Yaskawa INFORM job: A_ROOF_UPPER_0614_2_PAINT_10.JBI

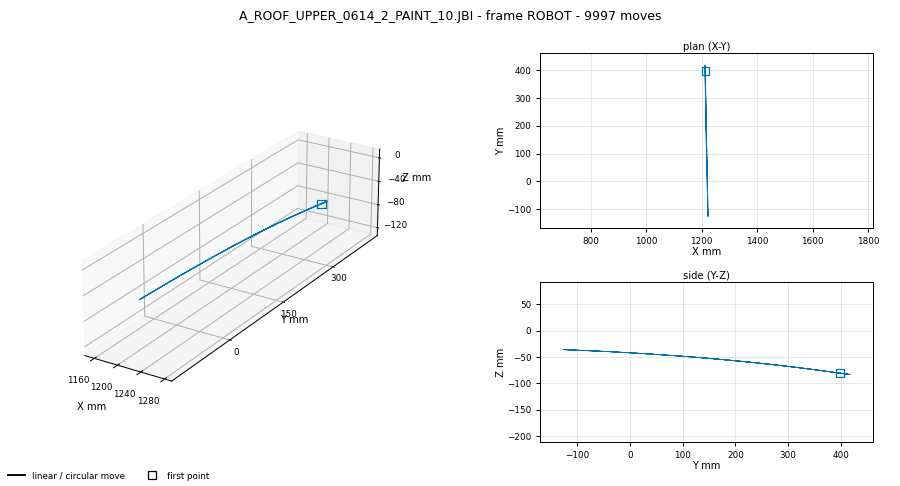
[picture p0: tool path of A_ROOF_UPPER_0614_2_PAINT_10.JBI in frame ROBOT, 9997 of 9997 moves have a stored position in this frame; points joined in program order, loops and branches not executed]
/JOB
//NAME A_ROOF_UPPER_0614_2_PAINT10
//POS
///NPOS 9997,0,0,0,0,0
///TOOL 1
///USER 0
///POSTYPE ROBOT
///RECTAN
///RCONF 1,0,0,0,0,0,0,0,0,0,0,0,0,0,0,0,0,0,0,0,0,0,0,0
C00000=1214.064,397.610,-80.249,-175.800,8.118,148.366
C00001=1214.059,397.858,-80.283,-175.800,8.120,148.367
C00002=1214.055,398.106,-80.318,-175.799,8.123,148.367
C00003=1214.051,398.353,-80.352,-175.799,8.125,148.368
C00004=1214.047,398.601,-80.386,-175.799,8.128,148.368
C00005=1214.043,398.849,-80.421,-175.797,8.130,148.369
C00006=1214.038,399.096,-80.456,-175.797,8.133,148.369
C00007=1214.035,399.343,-80.491,-175.796,8.135,148.370
C00008=1214.031,399.591,-80.525,-175.796,8.138,148.370
C00009=1214.027,399.839,-80.560,-175.795,8.140,148.371
C00010=1214.022,400.086,-80.594,-175.794,8.143,148.371
C00011=1214.019,400.334,-80.629,-175.794,8.145,148.372
C00012=1214.014,400.581,-80.663,-175.794,8.147,148.372
C00013=1214.010,400.830,-80.698,-175.793,8.150,148.373
C00014=1214.007,401.076,-80.732,-175.792,8.152,148.373
C00015=1214.003,401.324,-80.767,-175.792,8.154,148.373
C00016=1213.998,401.572,-80.802,-175.791,8.157,148.374
C00017=1213.994,401.819,-80.836,-175.791,8.159,148.374
C00018=1213.991,402.067,-80.870,-175.790,8.162,148.375
C00019=1213.986,402.314,-80.905,-175.790,8.164,148.375
C00020=1213.982,402.562,-80.940,-175.789,8.167,148.376
C00021=1213.978,402.809,-80.975,-175.788,8.169,148.376
C00022=1213.975,403.057,-81.009,-175.788,8.171,148.377
C00023=1213.970,403.304,-81.044,-175.787,8.174,148.377
C00024=1213.966,403.552,-81.079,-175.787,8.176,148.378
C00025=1213.962,403.799,-81.114,-175.787,8.178,148.378
C00026=1213.958,404.047,-81.149,-175.786,8.180,148.379
C00027=1213.954,404.295,-81.182,-175.785,8.183,148.379
C00028=1213.950,404.543,-81.217,-175.784,8.185,148.380
C00029=1213.946,404.789,-81.252,-175.784,8.188,148.380
C00030=1213.942,405.038,-81.287,-175.784,8.190,148.381
C00031=1213.937,405.285,-81.322,-175.783,8.192,148.381
C00032=1213.934,405.532,-81.357,-175.783,8.195,148.382
C00033=1213.930,405.780,-81.391,-175.782,8.197,148.382
C00034=1213.926,406.028,-81.426,-175.782,8.199,148.382
C00035=1213.921,406.275,-81.460,-175.782,8.202,148.383
C00036=1213.918,406.523,-81.496,-175.781,8.204,148.383
C00037=1213.914,406.770,-81.530,-175.780,8.207,148.384
C00038=1213.910,407.018,-81.565,-175.780,8.209,148.384
C00039=1213.905,407.265,-81.600,-175.779,8.211,148.385
C00040=1213.901,407.513,-81.635,-175.779,8.213,148.385
C00041=1213.897,407.760,-81.669,-175.778,8.215,148.386
C00042=1213.894,408.007,-81.704,-175.778,8.217,148.386
C00043=1213.890,408.256,-81.739,-175.777,8.220,148.387
C00044=1213.885,408.503,-81.773,-175.777,8.223,148.387
C00045=1213.882,408.750,-81.809,-175.776,8.224,148.387
C00046=1213.877,408.998,-81.843,-175.776,8.227,148.388
C00047=1213.873,409.246,-81.878,-175.776,8.229,148.388
C00048=1213.869,409.493,-81.913,-175.775,8.231,148.389
C00049=1213.866,409.741,-81.948,-175.775,8.233,148.389
C00050=1213.861,409.988,-81.982,-175.774,8.236,148.390
C00051=1213.858,410.236,-82.018,-175.774,8.238,148.390
C00052=1213.853,410.483,-82.052,-175.773,8.240,148.391
C00053=1213.849,410.730,-82.088,-175.773,8.243,148.391
C00054=1213.845,410.979,-82.123,-175.772,8.245,148.392
C00055=1213.841,411.226,-82.157,-175.772,8.247,148.392
C00056=1213.837,411.474,-82.193,-175.772,8.249,148.393
C00057=1213.833,411.721,-82.226,-175.771,8.251,148.393
C00058=1213.830,411.968,-82.262,-175.771,8.253,148.393
C00059=1213.825,412.216,-82.296,-175.770,8.255,148.394
C00060=1213.821,412.464,-82.331,-175.770,8.258,148.394
C00061=1213.817,412.710,-82.366,-175.770,8.260,148.395
C00062=1213.813,412.959,-82.401,-175.768,8.263,148.395
C00063=1213.809,413.206,-82.437,-175.768,8.265,148.396
C00064=1213.805,413.454,-82.471,-175.768,8.267,148.396
C00065=1213.801,413.701,-82.507,-175.767,8.269,148.397
C00066=1213.796,413.948,-82.541,-175.767,8.271,148.397
C00067=1213.793,414.196,-82.577,-175.767,8.273,148.398
C00068=1213.789,414.443,-82.611,-175.766,8.275,148.398
C00069=1213.785,414.691,-82.646,-175.766,8.278,148.398
C00070=1213.781,414.939,-82.681,-175.765,8.280,148.399
C00071=1213.777,415.186,-82.716,-175.765,8.282,148.399
C00072=1213.773,415.424,-82.750,-175.764,8.284,148.400
C00073=1213.769,415.662,-82.783,-175.764,8.286,148.400
C00074=1213.766,415.900,-82.817,-175.763,8.288,148.400
C00075=1213.761,416.139,-82.851,-175.763,8.290,148.401
C00076=1213.757,416.377,-82.885,-175.763,8.292,148.401
C00077=1213.754,416.616,-82.918,-175.763,8.294,148.402
C00078=1213.752,416.853,-82.951,-175.762,8.296,148.402
C00079=1213.753,417.091,-82.985,-175.762,8.298,148.403
C00080=1213.331,417.091,-83.021,-175.765,8.308,148.406
C00081=1213.330,416.852,-82.988,-175.765,8.306,148.406
C00082=1213.332,416.612,-82.954,-175.766,8.304,148.406
C00083=1213.336,416.372,-82.920,-175.766,8.302,148.405
C00084=1213.339,416.134,-82.886,-175.766,8.301,148.405
C00085=1213.343,415.894,-82.852,-175.767,8.299,148.404
C00086=1213.348,415.655,-82.818,-175.767,8.297,148.404
C00087=1213.351,415.415,-82.785,-175.768,8.295,148.403
C00088=1213.355,415.175,-82.750,-175.768,8.293,148.403
C00089=1213.359,414.928,-82.715,-175.768,8.290,148.402
C00090=1213.363,414.680,-82.680,-175.769,8.288,148.402
C00091=1213.367,414.433,-82.645,-175.769,8.286,148.402
C00092=1213.371,414.185,-82.610,-175.769,8.284,148.401
C00093=1213.376,413.938,-82.576,-175.770,8.282,148.401
C00094=1213.379,413.690,-82.540,-175.770,8.280,148.400
C00095=1213.383,413.442,-82.506,-175.771,8.278,148.400
C00096=1213.387,413.196,-82.471,-175.771,8.275,148.399
C00097=1213.391,412.947,-82.436,-175.772,8.273,148.399
C00098=1213.395,412.701,-82.401,-175.773,8.270,148.398
C00099=1213.399,412.453,-82.366,-175.773,8.268,148.398
C00100=1213.403,412.206,-82.331,-175.773,8.266,148.398
C00101=1213.407,411.958,-82.296,-175.774,8.264,148.397
C00102=1213.411,411.709,-82.261,-175.774,8.262,148.397
C00103=1213.416,411.463,-82.226,-175.775,8.259,148.396
C00104=1213.420,411.215,-82.191,-175.775,8.257,148.396
C00105=1213.424,410.968,-82.156,-175.775,8.255,148.395
C00106=1213.427,410.720,-82.122,-175.776,8.253,148.395
C00107=1213.431,410.473,-82.086,-175.776,8.251,148.394
C00108=1213.435,410.225,-82.052,-175.776,8.249,148.394
C00109=1213.439,409.977,-82.017,-175.777,8.247,148.393
C00110=1213.444,409.730,-81.982,-175.778,8.244,148.393
C00111=1213.447,409.482,-81.947,-175.779,8.242,148.393
C00112=1213.452,409.235,-81.912,-175.779,8.239,148.392
C00113=1213.455,408.987,-81.877,-175.779,8.237,148.391
C00114=1213.460,408.740,-81.843,-175.780,8.235,148.391
C00115=1213.463,408.492,-81.807,-175.780,8.233,148.391
C00116=1213.468,408.245,-81.773,-175.780,8.231,148.390
C00117=1213.472,407.997,-81.738,-175.781,8.229,148.390
C00118=1213.476,407.750,-81.703,-175.781,8.226,148.389
C00119=1213.480,407.502,-81.668,-175.782,8.224,148.389
C00120=1213.484,407.255,-81.634,-175.782,8.221,148.388
C00121=1213.487,407.007,-81.599,-175.783,8.219,148.388
C00122=1213.492,406.760,-81.564,-175.783,8.217,148.387
C00123=1213.496,406.512,-81.529,-175.783,8.215,148.387
C00124=1213.500,406.264,-81.494,-175.785,8.212,148.386
C00125=1213.504,406.017,-81.459,-175.785,8.210,148.386
C00126=1213.507,405.769,-81.425,-175.785,8.208,148.386
C00127=1213.512,405.522,-81.391,-175.786,8.205,148.385
C00128=1213.516,405.274,-81.355,-175.786,8.203,148.385
C00129=1213.520,405.027,-81.321,-175.787,8.200,148.384
C00130=1213.524,404.779,-81.286,-175.787,8.198,148.384
C00131=1213.528,404.532,-81.252,-175.788,8.196,148.383
C00132=1213.532,404.284,-81.216,-175.788,8.194,148.383
C00133=1213.536,404.037,-81.182,-175.789,8.191,148.382
C00134=1213.540,403.789,-81.147,-175.789,8.189,148.382
C00135=1213.544,403.541,-81.113,-175.790,8.186,148.381
C00136=1213.548,403.294,-81.078,-175.790,8.185,148.381
C00137=1213.552,403.046,-81.043,-175.791,8.181,148.380
C00138=1213.556,402.798,-81.008,-175.792,8.179,148.380
C00139=1213.561,402.551,-80.974,-175.792,8.177,148.379
C00140=1213.564,402.304,-80.939,-175.792,8.175,148.379
C00141=1213.568,402.056,-80.904,-175.793,8.172,148.379
C00142=1213.573,401.809,-80.870,-175.794,8.170,148.378
C00143=1213.577,401.561,-80.835,-175.794,8.168,148.378
C00144=1213.581,401.314,-80.801,-175.795,8.165,148.377
C00145=1213.584,401.066,-80.766,-175.795,8.162,148.377
C00146=1213.589,400.819,-80.731,-175.796,8.160,148.376
C00147=1213.593,400.571,-80.696,-175.797,8.157,148.376
C00148=1213.597,400.324,-80.663,-175.797,8.155,148.375
C00149=1213.601,400.075,-80.628,-175.797,8.153,148.375
C00150=1213.605,399.828,-80.593,-175.799,8.150,148.374
C00151=1213.609,399.580,-80.559,-175.799,8.148,148.374
C00152=1213.613,399.333,-80.524,-175.799,8.146,148.373
C00153=1213.617,399.085,-80.489,-175.800,8.143,148.373
C00154=1213.621,398.838,-80.455,-175.800,8.141,148.372
C00155=1213.625,398.591,-80.421,-175.801,8.139,148.372
C00156=1213.629,398.343,-80.386,-175.802,8.136,148.371
C00157=1213.634,398.095,-80.351,-175.802,8.133,148.371
C00158=1213.637,397.847,-80.317,-175.803,8.131,148.370
C00159=1213.642,397.600,-80.283,-175.803,8.128,148.370
C00160=1213.646,397.352,-80.248,-175.804,8.126,148.370
C00161=1213.650,397.105,-80.213,-175.805,8.123,148.369
C00162=1213.653,396.857,-80.178,-175.805,8.121,148.369
C00163=1213.658,396.610,-80.144,-175.806,8.118,148.368
C00164=1213.662,396.362,-80.109,-175.807,8.116,148.368
C00165=1213.665,396.115,-80.075,-175.808,8.113,148.367
C00166=1213.670,395.867,-80.041,-175.808,8.111,148.367
C00167=1213.674,395.619,-80.006,-175.808,8.109,148.366
C00168=1213.678,395.372,-79.972,-175.809,8.106,148.366
C00169=1213.682,395.125,-79.938,-175.810,8.104,148.365
C00170=1213.686,394.877,-79.903,-175.811,8.101,148.365
C00171=1213.690,394.629,-79.869,-175.811,8.099,148.364
C00172=1213.694,394.381,-79.834,-175.812,8.095,148.364
C00173=1213.698,394.134,-79.800,-175.813,8.094,148.363
C00174=1213.702,393.886,-79.765,-175.813,8.090,148.363
C00175=1213.706,393.639,-79.731,-175.814,8.088,148.362
C00176=1213.710,393.391,-79.697,-175.815,8.085,148.362
C00177=1213.715,393.108,-79.658,-175.816,8.082,148.361
C00178=1213.720,392.827,-79.618,-175.817,8.079,148.361
C00179=1213.724,392.544,-79.579,-175.817,8.076,148.360
C00180=1213.728,392.263,-79.541,-175.818,8.073,148.360
C00181=1213.733,392.015,-79.506,-175.819,8.071,148.359
C00182=1213.736,391.767,-79.472,-175.820,8.068,148.359
C00183=1213.741,391.520,-79.437,-175.820,8.066,148.358
C00184=1213.745,391.272,-79.403,-175.821,8.063,148.358
C00185=1213.749,391.025,-79.369,-175.822,8.061,148.357
C00186=1213.753,390.777,-79.334,-175.822,8.058,148.357
C00187=1213.756,390.529,-79.300,-175.824,8.055,148.356
C00188=1213.761,390.281,-79.266,-175.824,8.053,148.356
C00189=1213.765,390.034,-79.232,-175.825,8.050,148.356
C00190=1213.769,389.786,-79.197,-175.826,8.048,148.355
C00191=1213.774,389.539,-79.163,-175.826,8.045,148.355
C00192=1213.778,389.292,-79.129,-175.828,8.042,148.354
C00193=1213.781,389.043,-79.094,-175.828,8.040,148.354
C00194=1213.785,388.796,-79.060,-175.829,8.037,148.353
C00195=1213.790,388.548,-79.027,-175.830,8.034,148.353
C00196=1213.793,388.301,-78.992,-175.830,8.032,148.352
C00197=1213.798,388.053,-78.958,-175.831,8.029,148.352
C00198=1213.802,387.806,-78.924,-175.832,8.026,148.351
C00199=1213.806,387.558,-78.889,-175.833,8.024,148.351
C00200=1213.810,387.311,-78.855,-175.834,8.021,148.350
C00201=1213.815,387.063,-78.822,-175.835,8.018,148.350
C00202=1213.818,386.815,-78.787,-175.836,8.015,148.349
C00203=1213.822,386.568,-78.753,-175.836,8.013,148.349
C00204=1213.826,386.320,-78.719,-175.838,8.010,148.349
C00205=1213.830,386.072,-78.685,-175.838,8.007,148.348
C00206=1213.834,385.825,-78.651,-175.839,8.004,148.348
C00207=1213.839,385.577,-78.617,-175.840,8.002,148.347
C00208=1213.842,385.329,-78.582,-175.841,7.999,148.347
C00209=1213.847,385.081,-78.549,-175.842,7.996,148.346
C00210=1213.851,384.834,-78.515,-175.843,7.994,148.346
C00211=1213.854,384.586,-78.481,-175.843,7.991,148.345
C00212=1213.859,384.339,-78.446,-175.845,7.989,148.345
C00213=1213.863,384.091,-78.413,-175.846,7.986,148.345
C00214=1213.867,383.843,-78.378,-175.847,7.983,148.344
C00215=1213.870,383.596,-78.344,-175.848,7.980,148.344
C00216=1213.875,383.348,-78.310,-175.848,7.978,148.343
C00217=1213.879,383.101,-78.277,-175.849,7.975,148.343
C00218=1213.883,382.853,-78.242,-175.850,7.972,148.342
C00219=1213.887,382.605,-78.209,-175.852,7.969,148.342
C00220=1213.891,382.358,-78.175,-175.853,7.966,148.342
C00221=1213.896,382.110,-78.141,-175.853,7.963,148.341
C00222=1213.899,381.862,-78.107,-175.855,7.960,148.341
C00223=1213.904,381.615,-78.072,-175.855,7.958,148.340
C00224=1213.908,381.367,-78.039,-175.857,7.956,148.340
C00225=1213.911,381.119,-78.005,-175.857,7.952,148.339
C00226=1213.916,380.872,-77.970,-175.858,7.950,148.339
C00227=1213.920,380.624,-77.937,-175.860,7.947,148.338
C00228=1213.924,380.377,-77.903,-175.861,7.944,148.338
C00229=1213.928,380.128,-77.869,-175.862,7.941,148.337
C00230=1213.932,379.881,-77.835,-175.863,7.938,148.337
C00231=1213.937,379.633,-77.802,-175.864,7.935,148.337
C00232=1213.941,379.386,-77.768,-175.865,7.932,148.336
C00233=1213.945,379.138,-77.735,-175.866,7.930,148.336
C00234=1213.949,378.890,-77.700,-175.867,7.928,148.336
C00235=1213.953,378.642,-77.667,-175.868,7.925,148.335
C00236=1213.957,378.395,-77.633,-175.869,7.922,148.335
C00237=1213.961,378.147,-77.599,-175.870,7.919,148.334
C00238=1213.965,377.899,-77.565,-175.871,7.916,148.334
C00239=1213.969,377.652,-77.532,-175.873,7.913,148.333
C00240=1213.973,377.404,-77.498,-175.874,7.910,148.333
C00241=1213.978,377.156,-77.464,-175.875,7.908,148.333
C00242=1213.981,376.909,-77.430,-175.876,7.905,148.332
C00243=1213.985,376.661,-77.397,-175.877,7.902,148.332
C00244=1213.990,376.413,-77.362,-175.878,7.899,148.331
C00245=1213.994,376.166,-77.329,-175.879,7.896,148.331
C00246=1213.997,375.919,-77.295,-175.880,7.893,148.330
C00247=1214.002,375.671,-77.262,-175.882,7.890,148.330
C00248=1214.006,375.422,-77.228,-175.883,7.888,148.330
C00249=1214.010,375.175,-77.194,-175.884,7.885,148.329
C00250=1214.014,374.927,-77.161,-175.885,7.882,148.329
C00251=1214.018,374.680,-77.127,-175.887,7.878,148.328
C00252=1214.023,374.432,-77.093,-175.888,7.876,148.328
C00253=1214.026,374.184,-77.060,-175.889,7.873,148.328
C00254=1214.030,373.937,-77.026,-175.891,7.870,148.327
C00255=1214.034,373.689,-76.993,-175.892,7.867,148.327
C00256=1214.038,373.441,-76.959,-175.893,7.864,148.326
C00257=1214.043,373.194,-76.925,-175.894,7.861,148.326
C00258=1214.047,372.946,-76.892,-175.895,7.859,148.326
C00259=1214.050,372.698,-76.858,-175.897,7.856,148.325
C00260=1214.054,372.450,-76.824,-175.898,7.853,148.325
C00261=1214.058,372.203,-76.791,-175.899,7.851,148.325
C00262=1214.063,371.955,-76.758,-175.901,7.847,148.324
C00263=1214.067,371.707,-76.724,-175.902,7.844,148.324
C00264=1214.071,371.460,-76.691,-175.903,7.841,148.323
C00265=1214.075,371.212,-76.657,-175.905,7.838,148.323
C00266=1214.080,370.964,-76.624,-175.906,7.836,148.323
C00267=1214.083,370.716,-76.591,-175.907,7.833,148.322
C00268=1214.088,370.469,-76.556,-175.908,7.830,148.322
C00269=1214.092,370.221,-76.523,-175.910,7.827,148.322
C00270=1214.096,369.973,-76.490,-175.912,7.824,148.321
C00271=1214.100,369.725,-76.457,-175.913,7.821,148.321
C00272=1214.104,369.478,-76.424,-175.914,7.818,148.320
C00273=1214.108,369.231,-76.390,-175.915,7.815,148.320
C00274=1214.112,368.983,-76.357,-175.917,7.812,148.320
C00275=1214.116,368.735,-76.323,-175.919,7.809,148.319
C00276=1214.120,368.487,-76.290,-175.920,7.806,148.319
C00277=1214.125,368.239,-76.256,-175.921,7.804,148.319
C00278=1214.129,367.991,-76.223,-175.922,7.801,148.318
C00279=1214.133,367.743,-76.190,-175.924,7.797,148.318
C00280=1214.137,367.495,-76.157,-175.926,7.795,148.318
C00281=1214.142,367.216,-76.119,-175.927,7.792,148.317
C00282=1214.146,366.936,-76.081,-175.929,7.788,148.317
C00283=1214.151,366.656,-76.043,-175.931,7.785,148.317
C00284=1214.156,366.375,-76.006,-175.932,7.781,148.316
C00285=1214.160,366.127,-75.973,-175.934,7.778,148.316
C00286=1214.164,365.879,-75.940,-175.935,7.775,148.315
C00287=1214.168,365.632,-75.906,-175.936,7.773,148.315
C00288=1214.172,365.384,-75.873,-175.938,7.769,148.315
C00289=1214.176,365.136,-75.840,-175.940,7.767,148.315
C00290=1214.180,364.888,-75.807,-175.941,7.764,148.314
C00291=1214.184,364.641,-75.774,-175.942,7.761,148.314
C00292=1214.188,364.393,-75.741,-175.944,7.758,148.313
C00293=1214.193,364.145,-75.708,-175.946,7.755,148.313
C00294=1214.197,363.897,-75.674,-175.947,7.752,148.313
C00295=1214.201,363.650,-75.641,-175.949,7.749,148.312
C00296=1214.205,363.402,-75.608,-175.950,7.746,148.312
C00297=1214.209,363.154,-75.575,-175.952,7.743,148.312
C00298=1214.213,362.907,-75.542,-175.954,7.740,148.311
C00299=1214.217,362.659,-75.509,-175.955,7.737,148.311
C00300=1214.221,362.411,-75.476,-175.956,7.734,148.311
C00301=1214.225,362.164,-75.443,-175.959,7.731,148.311
C00302=1214.229,361.916,-75.410,-175.960,7.728,148.310
C00303=1214.233,361.668,-75.377,-175.961,7.726,148.310
C00304=1214.238,361.420,-75.344,-175.963,7.722,148.310
C00305=1214.242,361.172,-75.311,-175.965,7.720,148.309
C00306=1214.246,360.924,-75.278,-175.966,7.717,148.309
C00307=1214.250,360.677,-75.245,-175.968,7.713,148.309
C00308=1214.254,360.429,-75.212,-175.969,7.711,148.308
C00309=1214.258,360.181,-75.179,-175.971,7.708,148.308
C00310=1214.262,359.933,-75.147,-175.973,7.704,148.308
C00311=1214.266,359.685,-75.113,-175.974,7.702,148.308
C00312=1214.270,359.438,-75.080,-175.976,7.699,148.307
C00313=1214.275,359.190,-75.047,-175.978,7.696,148.307
C00314=1214.279,358.942,-75.015,-175.980,7.693,148.307
C00315=1214.283,358.694,-74.981,-175.982,7.690,148.307
C00316=1214.287,358.446,-74.949,-175.983,7.687,148.306
C00317=1214.291,358.199,-74.916,-175.985,7.685,148.306
C00318=1214.296,357.951,-74.884,-175.986,7.681,148.306
C00319=1214.300,357.703,-74.851,-175.988,7.678,148.305
C00320=1214.304,357.456,-74.817,-175.990,7.676,148.305
C00321=1214.308,357.208,-74.786,-175.991,7.672,148.305
C00322=1214.312,356.960,-74.752,-175.993,7.670,148.305
C00323=1214.316,356.712,-74.719,-175.995,7.666,148.304
C00324=1214.320,356.464,-74.687,-175.996,7.664,148.304
C00325=1214.325,356.216,-74.654,-175.998,7.661,148.304
C00326=1214.328,355.969,-74.621,-176.000,7.658,148.304
C00327=1214.332,355.720,-74.589,-176.002,7.655,148.303
C00328=1214.337,355.473,-74.555,-176.004,7.652,148.303
C00329=1214.342,355.225,-74.523,-176.005,7.649,148.303
C00330=1214.345,354.977,-74.491,-176.007,7.646,148.303
C00331=1214.349,354.730,-74.458,-176.009,7.643,148.302
C00332=1214.354,354.481,-74.425,-176.010,7.640,148.302
C00333=1214.357,354.234,-74.393,-176.012,7.637,148.302
C00334=1214.361,353.986,-74.360,-176.014,7.634,148.302
C00335=1214.366,353.738,-74.327,-176.016,7.631,148.301
C00336=1214.370,353.490,-74.295,-176.018,7.629,148.301
C00337=1214.374,353.243,-74.262,-176.019,7.626,148.301
C00338=1214.378,352.994,-74.230,-176.021,7.622,148.300
C00339=1214.383,352.747,-74.197,-176.023,7.620,148.300
C00340=1214.386,352.499,-74.165,-176.025,7.617,148.300
C00341=1214.390,352.251,-74.132,-176.027,7.614,148.300
C00342=1214.395,352.003,-74.099,-176.028,7.612,148.300
C00343=1214.399,351.756,-74.067,-176.030,7.608,148.299
C00344=1214.403,351.508,-74.035,-176.032,7.605,148.299
C00345=1214.407,351.260,-74.002,-176.034,7.602,148.299
C00346=1214.411,351.012,-73.970,-176.036,7.599,148.299
C00347=1214.416,350.763,-73.937,-176.038,7.596,148.298
C00348=1214.419,350.516,-73.905,-176.040,7.594,148.298
C00349=1214.424,350.268,-73.873,-176.042,7.590,148.298
C00350=1214.428,350.020,-73.840,-176.043,7.588,148.298
C00351=1214.432,349.773,-73.808,-176.045,7.585,148.298
C00352=1214.436,349.524,-73.775,-176.047,7.582,148.297
C00353=1214.441,349.277,-73.744,-176.048,7.579,148.297
C00354=1214.445,349.029,-73.711,-176.051,7.576,148.297
C00355=1214.449,348.781,-73.678,-176.052,7.573,148.297
C00356=1214.453,348.533,-73.646,-176.054,7.570,148.296
C00357=1214.457,348.285,-73.613,-176.056,7.567,148.296
C00358=1214.461,348.038,-73.582,-176.058,7.564,148.296
C00359=1214.466,347.789,-73.549,-176.060,7.561,148.296
C00360=1214.470,347.541,-73.517,-176.062,7.559,148.296
C00361=1214.474,347.294,-73.484,-176.064,7.556,148.295
C00362=1214.478,347.046,-73.453,-176.065,7.553,148.295
C00363=1214.482,346.798,-73.420,-176.068,7.550,148.295
C00364=1214.486,346.550,-73.388,-176.069,7.547,148.295
C00365=1214.490,346.302,-73.355,-176.072,7.544,148.295
C00366=1214.495,346.055,-73.324,-176.073,7.541,148.294
C00367=1214.499,345.806,-73.291,-176.075,7.538,148.294
C00368=1214.503,345.558,-73.260,-176.077,7.535,148.294
C00369=1214.508,345.311,-73.227,-176.080,7.532,148.294
C00370=1214.511,345.063,-73.196,-176.081,7.530,148.294
C00371=1214.516,344.815,-73.162,-176.084,7.527,148.294
C00372=1214.519,344.567,-73.131,-176.085,7.524,148.293
C00373=1214.524,344.319,-73.099,-176.087,7.521,148.293
C00374=1214.528,344.071,-73.067,-176.089,7.518,148.293
C00375=1214.532,343.823,-73.034,-176.091,7.516,148.293
C00376=1214.537,343.576,-73.003,-176.093,7.512,148.293
C00377=1214.540,343.328,-72.971,-176.095,7.510,148.292
C00378=1214.545,343.079,-72.938,-176.097,7.506,148.292
C00379=1214.549,342.832,-72.907,-176.099,7.504,148.292
C00380=1214.554,342.584,-72.875,-176.101,7.501,148.292
C00381=1214.557,342.335,-72.843,-176.103,7.498,148.292
C00382=1214.562,342.088,-72.811,-176.105,7.495,148.292
C00383=1214.566,341.840,-72.779,-176.107,7.492,148.291
C00384=1214.570,341.592,-72.747,-176.109,7.489,148.291
C00385=1214.575,341.314,-72.711,-176.111,7.486,148.291
C00386=1214.579,341.036,-72.675,-176.114,7.483,148.291
C00387=1214.585,340.758,-72.640,-176.115,7.480,148.291
C00388=1214.589,340.480,-72.604,-176.117,7.477,148.291
C00389=1214.593,340.232,-72.572,-176.120,7.473,148.290
C00390=1214.597,339.984,-72.540,-176.122,7.471,148.290
C00391=1214.601,339.737,-72.508,-176.124,7.468,148.290
C00392=1214.605,339.489,-72.476,-176.126,7.465,148.290
C00393=1214.610,339.240,-72.445,-176.128,7.462,148.290
C00394=1214.614,338.992,-72.413,-176.130,7.460,148.290
C00395=1214.618,338.744,-72.381,-176.132,7.456,148.290
C00396=1214.622,338.497,-72.350,-176.134,7.454,148.289
C00397=1214.627,338.249,-72.317,-176.136,7.451,148.289
C00398=1214.631,338.001,-72.286,-176.138,7.448,148.289
C00399=1214.635,337.753,-72.254,-176.140,7.445,148.289
C00400=1214.639,337.505,-72.223,-176.142,7.442,148.289
C00401=1214.644,337.257,-72.191,-176.145,7.439,148.289
C00402=1214.647,337.009,-72.159,-176.146,7.437,148.289
C00403=1214.652,336.762,-72.128,-176.148,7.434,148.288
C00404=1214.656,336.513,-72.097,-176.150,7.431,148.288
C00405=1214.660,336.265,-72.064,-176.153,7.428,148.288
C00406=1214.664,336.017,-72.033,-176.154,7.425,148.288
C00407=1214.668,335.769,-72.001,-176.157,7.422,148.288
C00408=1214.673,335.521,-71.970,-176.159,7.420,148.288
C00409=1214.676,335.273,-71.938,-176.161,7.417,148.288
C00410=1214.681,335.026,-71.907,-176.163,7.414,148.288
C00411=1214.686,334.777,-71.875,-176.165,7.411,148.287
C00412=1214.690,334.529,-71.843,-176.167,7.408,148.287
C00413=1214.694,334.281,-71.812,-176.169,7.405,148.287
C00414=1214.698,334.033,-71.781,-176.171,7.403,148.287
C00415=1214.702,333.785,-71.749,-176.173,7.400,148.287
C00416=1214.706,333.537,-71.717,-176.175,7.397,148.287
C00417=1214.710,333.289,-71.686,-176.178,7.394,148.287
C00418=1214.714,333.041,-71.655,-176.180,7.392,148.287
C00419=1214.719,332.793,-71.623,-176.182,7.388,148.287
C00420=1214.723,332.545,-71.591,-176.184,7.386,148.286
C00421=1214.728,332.297,-71.561,-176.186,7.383,148.286
C00422=1214.731,332.049,-71.529,-176.188,7.380,148.286
C00423=1214.736,331.802,-71.497,-176.191,7.377,148.286
C00424=1214.740,331.554,-71.466,-176.192,7.375,148.286
C00425=1214.744,331.306,-71.435,-176.195,7.372,148.286
C00426=1214.749,331.058,-71.404,-176.197,7.369,148.286
C00427=1214.752,330.810,-71.372,-176.199,7.366,148.286
C00428=1214.757,330.562,-71.341,-176.201,7.364,148.286
C00429=1214.761,330.314,-71.309,-176.203,7.360,148.285
C00430=1214.765,330.066,-71.279,-176.205,7.358,148.285
C00431=1214.769,329.817,-71.248,-176.207,7.355,148.285
C00432=1214.773,329.570,-71.216,-176.209,7.353,148.285
C00433=1214.777,329.321,-71.185,-176.212,7.349,148.285
C00434=1214.782,329.074,-71.153,-176.214,7.347,148.285
C00435=1214.786,328.825,-71.122,-176.216,7.344,148.285
C00436=1214.790,328.577,-71.092,-176.218,7.341,148.285
C00437=1214.795,328.330,-71.060,-176.220,7.338,148.285
C00438=1214.799,328.081,-71.029,-176.222,7.336,148.285
C00439=1214.803,327.834,-70.997,-176.225,7.333,148.285
C00440=1214.807,327.585,-70.966,-176.227,7.330,148.285
C00441=1214.812,327.337,-70.936,-176.229,7.327,148.285
C00442=1214.816,327.089,-70.905,-176.231,7.325,148.284
C00443=1214.820,326.841,-70.873,-176.234,7.322,148.284
C00444=1214.825,326.593,-70.842,-176.235,7.319,148.284
C00445=1214.829,326.345,-70.811,-176.238,7.316,148.284
C00446=1214.833,326.097,-70.780,-176.240,7.314,148.284
C00447=1214.837,325.850,-70.749,-176.242,7.311,148.284
C00448=1214.841,325.601,-70.718,-176.244,7.308,148.284
C00449=1214.845,325.353,-70.688,-176.247,7.305,148.284
C00450=1214.849,325.105,-70.656,-176.249,7.303,148.284
C00451=1214.854,324.857,-70.625,-176.251,7.299,148.284
C00452=1214.858,324.609,-70.594,-176.253,7.297,148.284
C00453=1214.862,324.360,-70.563,-176.256,7.294,148.284
C00454=1214.866,324.113,-70.533,-176.257,7.292,148.284
C00455=1214.871,323.865,-70.501,-176.260,7.289,148.284
C00456=1214.875,323.617,-70.470,-176.262,7.286,148.284
C00457=1214.879,323.369,-70.439,-176.264,7.283,148.283
C00458=1214.884,323.121,-70.409,-176.266,7.281,148.283
C00459=1214.887,322.873,-70.378,-176.269,7.277,148.283
C00460=1214.892,322.625,-70.347,-176.271,7.275,148.283
C00461=1214.896,322.377,-70.317,-176.273,7.272,148.283
C00462=1214.900,322.128,-70.286,-176.275,7.270,148.283
C00463=1214.904,321.880,-70.255,-176.278,7.267,148.283
C00464=1214.909,321.632,-70.225,-176.280,7.264,148.283
C00465=1214.912,321.384,-70.193,-176.282,7.261,148.283
C00466=1214.917,321.136,-70.162,-176.284,7.259,148.283
C00467=1214.921,320.889,-70.132,-176.287,7.256,148.283
C00468=1214.925,320.640,-70.101,-176.289,7.254,148.283
C00469=1214.930,320.392,-70.070,-176.291,7.250,148.283
C00470=1214.934,320.144,-70.039,-176.293,7.248,148.283
C00471=1214.938,319.896,-70.009,-176.296,7.245,148.283
C00472=1214.942,319.648,-69.978,-176.298,7.243,148.283
C00473=1214.947,319.399,-69.948,-176.300,7.239,148.283
C00474=1214.951,319.152,-69.918,-176.302,7.237,148.283
C00475=1214.956,318.904,-69.887,-176.305,7.234,148.283
C00476=1214.960,318.655,-69.856,-176.307,7.232,148.283
C00477=1214.963,318.407,-69.826,-176.309,7.229,148.283
C00478=1214.968,318.159,-69.795,-176.311,7.226,148.283
C00479=1214.973,317.911,-69.764,-176.314,7.223,148.283
C00480=1214.976,317.663,-69.734,-176.316,7.221,148.282
C00481=1214.981,317.415,-69.703,-176.318,7.218,148.282
C00482=1214.985,317.167,-69.673,-176.321,7.216,148.282
C00483=1214.989,316.919,-69.643,-176.323,7.213,148.282
C00484=1214.993,316.670,-69.611,-176.325,7.210,148.282
C00485=1214.997,316.423,-69.581,-176.328,7.207,148.282
C00486=1215.002,316.175,-69.550,-176.330,7.205,148.282
C00487=1215.006,315.927,-69.520,-176.332,7.202,148.282
C00488=1215.011,315.678,-69.490,-176.334,7.200,148.282
C00489=1215.015,315.403,-69.456,-176.337,7.196,148.282
C00490=1215.020,315.126,-69.422,-176.339,7.193,148.282
C00491=1215.025,314.851,-69.389,-176.342,7.190,148.282
C00492=1215.029,314.575,-69.354,-176.345,7.187,148.282
C00493=1215.034,314.326,-69.324,-176.347,7.185,148.282
C00494=1215.037,314.078,-69.294,-176.349,7.182,148.282
C00495=1215.042,313.830,-69.263,-176.352,7.180,148.282
C00496=1215.046,313.582,-69.234,-176.354,7.177,148.282
C00497=1215.051,313.334,-69.203,-176.356,7.174,148.282
C00498=1215.055,313.086,-69.173,-176.359,7.171,148.282
C00499=1215.060,312.838,-69.143,-176.361,7.169,148.282
C00500=1215.063,312.589,-69.112,-176.363,7.166,148.282
C00501=1215.068,312.341,-69.082,-176.365,7.164,148.282
C00502=1215.072,312.093,-69.052,-176.368,7.161,148.282
C00503=1215.076,311.845,-69.021,-176.370,7.158,148.282
C00504=1215.081,311.597,-68.992,-176.372,7.155,148.282
C00505=1215.085,311.349,-68.961,-176.375,7.153,148.282
C00506=1215.089,311.101,-68.931,-176.377,7.150,148.282
C00507=1215.094,310.853,-68.901,-176.379,7.147,148.282
C00508=1215.098,310.604,-68.871,-176.382,7.144,148.282
C00509=1215.101,310.356,-68.841,-176.384,7.142,148.282
C00510=1215.106,310.107,-68.811,-176.387,7.139,148.282
C00511=1215.110,309.860,-68.780,-176.389,7.137,148.282
C00512=1215.115,309.611,-68.750,-176.392,7.134,148.282
C00513=1215.119,309.364,-68.720,-176.394,7.132,148.282
C00514=1215.123,309.115,-68.691,-176.396,7.128,148.282
C00515=1215.128,308.867,-68.660,-176.398,7.126,148.282
C00516=1215.132,308.619,-68.631,-176.401,7.123,148.282
C00517=1215.136,308.371,-68.600,-176.403,7.121,148.282
C00518=1215.141,308.123,-68.570,-176.405,7.118,148.282
C00519=1215.145,307.875,-68.541,-176.408,7.116,148.282
C00520=1215.150,307.627,-68.510,-176.410,7.113,148.282
C00521=1215.154,307.378,-68.481,-176.412,7.110,148.282
C00522=1215.158,307.131,-68.451,-176.415,7.108,148.282
C00523=1215.162,306.882,-68.421,-176.417,7.105,148.282
C00524=1215.167,306.634,-68.391,-176.419,7.103,148.283
C00525=1215.171,306.386,-68.361,-176.422,7.100,148.283
C00526=1215.175,306.138,-68.331,-176.424,7.098,148.283
C00527=1215.180,305.889,-68.301,-176.427,7.095,148.283
C00528=1215.184,305.642,-68.271,-176.429,7.092,148.283
C00529=1215.188,305.393,-68.242,-176.432,7.089,148.283
C00530=1215.193,305.145,-68.212,-176.434,7.087,148.283
C00531=1215.197,304.897,-68.182,-176.436,7.084,148.283
C00532=1215.201,304.649,-68.152,-176.438,7.082,148.283
C00533=1215.205,304.401,-68.123,-176.441,7.079,148.283
C00534=1215.209,304.152,-68.093,-176.443,7.077,148.283
C00535=1215.214,303.904,-68.063,-176.445,7.075,148.283
C00536=1215.218,303.656,-68.034,-176.448,7.072,148.283
C00537=1215.222,303.408,-68.004,-176.450,7.069,148.283
C00538=1215.226,303.160,-67.974,-176.453,7.066,148.283
C00539=1215.231,302.911,-67.944,-176.455,7.064,148.283
C00540=1215.235,302.663,-67.915,-176.458,7.061,148.283
C00541=1215.240,302.415,-67.885,-176.460,7.059,148.283
C00542=1215.244,302.166,-67.856,-176.462,7.056,148.283
C00543=1215.248,301.918,-67.826,-176.465,7.054,148.283
C00544=1215.252,301.670,-67.796,-176.467,7.051,148.283
C00545=1215.257,301.422,-67.766,-176.469,7.048,148.283
C00546=1215.261,301.174,-67.737,-176.471,7.046,148.283
C00547=1215.265,300.925,-67.707,-176.474,7.043,148.283
C00548=1215.269,300.677,-67.678,-176.477,7.041,148.284
C00549=1215.273,300.429,-67.648,-176.479,7.038,148.284
C00550=1215.278,300.180,-67.619,-176.482,7.036,148.284
C00551=1215.282,299.933,-67.590,-176.484,7.033,148.284
C00552=1215.287,299.685,-67.560,-176.486,7.031,148.284
C00553=1215.291,299.436,-67.531,-176.489,7.028,148.284
C00554=1215.295,299.188,-67.501,-176.491,7.025,148.284
C00555=1215.300,298.939,-67.471,-176.493,7.023,148.284
C00556=1215.304,298.691,-67.442,-176.496,7.020,148.284
C00557=1215.308,298.443,-67.412,-176.498,7.018,148.284
C00558=1215.312,298.195,-67.383,-176.501,7.015,148.284
C00559=1215.317,297.947,-67.354,-176.503,7.013,148.284
C00560=1215.321,297.699,-67.324,-176.506,7.010,148.284
C00561=1215.326,297.450,-67.296,-176.508,7.008,148.284
C00562=1215.330,297.202,-67.266,-176.511,7.005,148.284
C00563=1215.334,296.953,-67.237,-176.513,7.003,148.284
C00564=1215.338,296.705,-67.207,-176.515,7.000,148.284
C00565=1215.343,296.457,-67.178,-176.518,6.997,148.284
C00566=1215.347,296.209,-67.149,-176.520,6.995,148.285
C00567=1215.352,295.961,-67.119,-176.523,6.992,148.285
C00568=1215.356,295.712,-67.090,-176.525,6.990,148.285
C00569=1215.360,295.464,-67.061,-176.528,6.987,148.285
C00570=1215.364,295.216,-67.032,-176.530,6.985,148.285
C00571=1215.368,294.968,-67.003,-176.532,6.983,148.285
C00572=1215.373,294.720,-66.974,-176.535,6.980,148.285
C00573=1215.377,294.471,-66.945,-176.537,6.978,148.285
C00574=1215.381,294.223,-66.915,-176.540,6.975,148.285
C00575=1215.385,293.975,-66.886,-176.542,6.973,148.285
C00576=1215.390,293.726,-66.857,-176.544,6.970,148.285
C00577=1215.395,293.478,-66.828,-176.547,6.967,148.285
C00578=1215.399,293.230,-66.799,-176.549,6.965,148.286
C00579=1215.403,292.982,-66.769,-176.552,6.962,148.286
C00580=1215.408,292.733,-66.741,-176.554,6.960,148.286
C00581=1215.411,292.485,-66.712,-176.557,6.957,148.286
C00582=1215.416,292.237,-66.683,-176.559,6.955,148.286
C00583=1215.420,291.988,-66.654,-176.561,6.953,148.286
C00584=1215.424,291.740,-66.624,-176.564,6.950,148.286
C00585=1215.429,291.492,-66.595,-176.566,6.948,148.286
C00586=1215.434,291.244,-66.567,-176.569,6.945,148.286
C00587=1215.437,290.996,-66.538,-176.571,6.943,148.286
C00588=1215.442,290.747,-66.509,-176.573,6.940,148.286
C00589=1215.446,290.499,-66.480,-176.577,6.938,148.287
C00590=1215.451,290.250,-66.451,-176.579,6.936,148.287
C00591=1215.455,290.002,-66.422,-176.581,6.932,148.287
C00592=1215.459,289.754,-66.393,-176.583,6.930,148.287
C00593=1215.463,289.480,-66.361,-176.587,6.928,148.287
C00594=1215.469,289.205,-66.329,-176.589,6.925,148.287
C00595=1215.474,288.931,-66.297,-176.591,6.922,148.287
C00596=1215.478,288.657,-66.265,-176.595,6.920,148.287
C00597=1215.483,288.409,-66.237,-176.597,6.917,148.287
C00598=1215.487,288.161,-66.208,-176.599,6.914,148.287
C00599=1215.491,287.912,-66.179,-176.602,6.912,148.288
C00600=1215.496,287.664,-66.151,-176.605,6.909,148.288
C00601=1215.500,287.416,-66.122,-176.607,6.907,148.288
C00602=1215.504,287.167,-66.093,-176.609,6.905,148.288
C00603=1215.509,286.919,-66.064,-176.612,6.902,148.288
C00604=1215.513,286.671,-66.036,-176.614,6.900,148.288
C00605=1215.517,286.422,-66.007,-176.616,6.898,148.288
C00606=1215.522,286.174,-65.978,-176.619,6.895,148.288
C00607=1215.526,285.926,-65.950,-176.622,6.893,148.289
C00608=1215.530,285.677,-65.921,-176.624,6.890,148.289
C00609=1215.535,285.429,-65.892,-176.626,6.888,148.289
C00610=1215.539,285.181,-65.864,-176.629,6.886,148.289
C00611=1215.544,284.933,-65.835,-176.632,6.883,148.289
C00612=1215.548,284.684,-65.806,-176.634,6.881,148.289
C00613=1215.552,284.436,-65.778,-176.636,6.878,148.289
C00614=1215.557,284.188,-65.750,-176.639,6.876,148.289
C00615=1215.560,283.940,-65.721,-176.641,6.874,148.289
C00616=1215.565,283.691,-65.692,-176.643,6.871,148.289
C00617=1215.570,283.443,-65.664,-176.646,6.869,148.290
C00618=1215.574,283.194,-65.635,-176.649,6.866,148.290
C00619=1215.579,282.946,-65.607,-176.651,6.863,148.290
C00620=1215.582,282.698,-65.578,-176.654,6.861,148.290
C00621=1215.587,282.450,-65.550,-176.656,6.859,148.290
C00622=1215.591,282.201,-65.522,-176.659,6.856,148.290
C00623=1215.596,281.952,-65.493,-176.661,6.854,148.290
C00624=1215.601,281.704,-65.465,-176.663,6.852,148.291
C00625=1215.604,281.455,-65.436,-176.666,6.849,148.291
C00626=1215.609,281.208,-65.407,-176.669,6.847,148.291
C00627=1215.613,280.959,-65.379,-176.671,6.845,148.291
C00628=1215.618,280.711,-65.351,-176.673,6.842,148.291
C00629=1215.622,280.462,-65.323,-176.676,6.840,148.291
C00630=1215.627,280.214,-65.294,-176.678,6.838,148.291
C00631=1215.631,279.966,-65.266,-176.681,6.835,148.291
C00632=1215.635,279.718,-65.238,-176.684,6.833,148.292
C00633=1215.639,279.469,-65.210,-176.686,6.831,148.292
C00634=1215.643,279.220,-65.181,-176.688,6.828,148.292
C00635=1215.648,278.972,-65.153,-176.691,6.826,148.292
C00636=1215.652,278.724,-65.125,-176.693,6.824,148.292
C00637=1215.657,278.475,-65.097,-176.696,6.821,148.292
C00638=1215.661,278.227,-65.068,-176.698,6.819,148.292
C00639=1215.666,277.979,-65.040,-176.700,6.817,148.292
C00640=1215.670,277.730,-65.012,-176.704,6.814,148.293
C00641=1215.674,277.482,-64.984,-176.706,6.812,148.293
C00642=1215.679,277.233,-64.955,-176.708,6.809,148.293
C00643=1215.683,276.985,-64.928,-176.711,6.807,148.293
C00644=1215.687,276.738,-64.900,-176.713,6.805,148.293
C00645=1215.692,276.489,-64.871,-176.716,6.803,148.294
C00646=1215.696,276.241,-64.843,-176.718,6.800,148.294
C00647=1215.701,275.992,-64.815,-176.721,6.797,148.294
C00648=1215.705,275.743,-64.788,-176.723,6.796,148.294
C00649=1215.709,275.495,-64.759,-176.726,6.793,148.294
C00650=1215.714,275.247,-64.731,-176.728,6.791,148.294
C00651=1215.718,274.998,-64.703,-176.731,6.788,148.294
C00652=1215.722,274.750,-64.675,-176.733,6.785,148.294
C00653=1215.727,274.501,-64.646,-176.736,6.784,148.295
C00654=1215.731,274.253,-64.619,-176.738,6.781,148.295
C00655=1215.736,274.005,-64.592,-176.741,6.779,148.295
C00656=1215.739,273.756,-64.563,-176.743,6.776,148.295
C00657=1215.745,273.508,-64.535,-176.746,6.775,148.295
C00658=1215.749,273.259,-64.508,-176.748,6.772,148.295
C00659=1215.753,273.011,-64.480,-176.751,6.769,148.295
C00660=1215.757,272.763,-64.452,-176.753,6.767,148.296
C00661=1215.762,272.514,-64.423,-176.755,6.765,148.296
C00662=1215.766,272.266,-64.396,-176.758,6.763,148.296
C00663=1215.770,272.017,-64.368,-176.761,6.760,148.296
C00664=1215.775,271.769,-64.340,-176.763,6.758,148.296
C00665=1215.780,271.521,-64.313,-176.765,6.756,148.296
C00666=1215.784,271.272,-64.285,-176.769,6.754,148.297
C00667=1215.788,271.024,-64.257,-176.771,6.751,148.297
C00668=1215.793,270.776,-64.230,-176.773,6.749,148.297
C00669=1215.796,270.527,-64.202,-176.776,6.747,148.297
C00670=1215.802,270.279,-64.173,-176.778,6.744,148.297
C00671=1215.806,270.030,-64.146,-176.781,6.742,148.298
C00672=1215.810,269.782,-64.118,-176.783,6.740,148.298
C00673=1215.815,269.533,-64.091,-176.786,6.737,148.298
C00674=1215.818,269.285,-64.063,-176.788,6.735,148.298
C00675=1215.823,269.036,-64.036,-176.791,6.733,148.298
C00676=1215.828,268.788,-64.007,-176.793,6.731,148.298
C00677=1215.832,268.539,-63.979,-176.796,6.728,148.299
C00678=1215.836,268.291,-63.952,-176.798,6.726,148.299
C00679=1215.841,268.043,-63.924,-176.801,6.724,148.299
C00680=1215.845,267.795,-63.897,-176.803,6.722,148.299
C00681=1215.849,267.546,-63.869,-176.806,6.720,148.299
C00682=1215.854,267.298,-63.842,-176.808,6.717,148.299
C00683=1215.858,267.050,-63.814,-176.811,6.715,148.300
C00684=1215.862,266.800,-63.787,-176.814,6.712,148.300
C00685=1215.867,266.552,-63.760,-176.816,6.711,148.300
C00686=1215.872,266.304,-63.731,-176.818,6.708,148.300
C00687=1215.877,266.055,-63.704,-176.821,6.706,148.300
C00688=1215.880,265.807,-63.676,-176.824,6.703,148.300
C00689=1215.885,265.558,-63.649,-176.826,6.702,148.301
C00690=1215.890,265.310,-63.622,-176.828,6.699,148.301
C00691=1215.894,265.062,-63.594,-176.831,6.697,148.301
C00692=1215.898,264.813,-63.567,-176.833,6.695,148.301
C00693=1215.903,264.564,-63.540,-176.836,6.693,148.301
C00694=1215.907,264.316,-63.512,-176.838,6.690,148.301
C00695=1215.912,264.068,-63.485,-176.841,6.689,148.302
C00696=1215.916,263.819,-63.458,-176.843,6.686,148.302
C00697=1215.920,263.546,-63.428,-176.846,6.684,148.302
C00698=1215.926,263.274,-63.398,-176.849,6.681,148.302
C00699=1215.930,263.001,-63.368,-176.852,6.679,148.302
C00700=1215.935,262.729,-63.338,-176.855,6.676,148.303
C00701=1215.940,262.480,-63.310,-176.857,6.674,148.303
C00702=1215.944,262.231,-63.283,-176.860,6.672,148.303
C00703=1215.949,261.983,-63.255,-176.862,6.670,148.303
C00704=1215.952,261.735,-63.229,-176.865,6.667,148.303
C00705=1215.957,261.487,-63.202,-176.867,6.665,148.304
C00706=1215.961,261.237,-63.174,-176.870,6.663,148.304
C00707=1215.966,260.989,-63.147,-176.872,6.661,148.304
C00708=1215.970,260.741,-63.119,-176.874,6.659,148.304
C00709=1215.975,260.492,-63.092,-176.877,6.656,148.304
C00710=1215.979,260.244,-63.065,-176.880,6.654,148.305
C00711=1215.984,259.995,-63.038,-176.882,6.652,148.305
C00712=1215.988,259.746,-63.011,-176.885,6.650,148.305
C00713=1215.992,259.498,-62.984,-176.887,6.648,148.305
C00714=1215.997,259.250,-62.957,-176.890,6.645,148.306
C00715=1216.001,259.001,-62.930,-176.892,6.643,148.306
C00716=1216.006,258.753,-62.903,-176.895,6.641,148.306
C00717=1216.010,258.505,-62.875,-176.898,6.639,148.306
C00718=1216.015,258.256,-62.848,-176.900,6.637,148.306
C00719=1216.018,258.007,-62.822,-176.903,6.635,148.307
C00720=1216.023,257.759,-62.794,-176.905,6.632,148.307
C00721=1216.028,257.510,-62.767,-176.908,6.630,148.307
C00722=1216.032,257.262,-62.740,-176.910,6.628,148.307
C00723=1216.037,257.013,-62.713,-176.912,6.626,148.307
C00724=1216.041,256.765,-62.687,-176.915,6.624,148.308
C00725=1216.046,256.517,-62.660,-176.918,6.622,148.308
C00726=1216.050,256.268,-62.633,-176.920,6.620,148.308
C00727=1216.055,256.020,-62.606,-176.922,6.617,148.308
C00728=1216.058,255.771,-62.579,-176.925,6.616,148.308
C00729=1216.063,255.522,-62.552,-176.928,6.613,148.309
C00730=1216.068,255.273,-62.525,-176.930,6.611,148.309
C00731=1216.072,255.025,-62.499,-176.933,6.609,148.309
C00732=1216.076,254.776,-62.472,-176.935,6.607,148.309
C00733=1216.081,254.528,-62.445,-176.938,6.605,148.309
C00734=1216.086,254.279,-62.418,-176.940,6.603,148.310
C00735=1216.090,254.031,-62.391,-176.943,6.600,148.310
C00736=1216.094,253.783,-62.364,-176.946,6.598,148.310
C00737=1216.099,253.534,-62.337,-176.948,6.596,148.310
C00738=1216.103,253.286,-62.311,-176.950,6.594,148.310
C00739=1216.108,253.037,-62.284,-176.953,6.592,148.311
C00740=1216.113,252.789,-62.257,-176.955,6.590,148.311
C00741=1216.116,252.540,-62.231,-176.958,6.587,148.311
C00742=1216.121,252.292,-62.204,-176.961,6.585,148.311
C00743=1216.125,252.043,-62.178,-176.963,6.583,148.312
C00744=1216.130,251.795,-62.151,-176.966,6.581,148.312
C00745=1216.135,251.546,-62.124,-176.968,6.579,148.312
C00746=1216.139,251.298,-62.097,-176.970,6.577,148.312
C00747=1216.144,251.049,-62.071,-176.974,6.574,148.313
C00748=1216.147,250.801,-62.045,-176.976,6.573,148.313
C00749=1216.152,250.552,-62.018,-176.978,6.570,148.313
C00750=1216.157,250.303,-61.991,-176.981,6.569,148.313
C00751=1216.161,250.055,-61.965,-176.983,6.566,148.313
C00752=1216.166,249.806,-61.938,-176.986,6.565,148.314
C00753=1216.170,249.557,-61.912,-176.988,6.563,148.314
C00754=1216.175,249.309,-61.885,-176.991,6.560,148.314
C00755=1216.178,249.061,-61.858,-176.994,6.558,148.314
C00756=1216.183,248.812,-61.832,-176.996,6.556,148.315
C00757=1216.187,248.563,-61.806,-176.998,6.554,148.315
C00758=1216.192,248.314,-61.779,-177.001,6.552,148.315
C00759=1216.196,248.066,-61.753,-177.004,6.550,148.315
C00760=1216.201,247.818,-61.726,-177.006,6.548,148.315
C00761=1216.205,247.569,-61.700,-177.009,6.545,148.316
C00762=1216.210,247.320,-61.673,-177.012,6.543,148.316
C00763=1216.214,247.072,-61.647,-177.014,6.541,148.316
C00764=1216.219,246.823,-61.620,-177.016,6.539,148.316
C00765=1216.223,246.575,-61.595,-177.019,6.537,148.317
C00766=1216.228,246.326,-61.568,-177.022,6.535,148.317
C00767=1216.232,246.078,-61.542,-177.024,6.533,148.317
C00768=1216.237,245.829,-61.515,-177.026,6.531,148.317
C00769=1216.241,245.580,-61.489,-177.029,6.529,148.318
C00770=1216.246,245.332,-61.462,-177.032,6.526,148.318
C00771=1216.250,245.083,-61.436,-177.034,6.525,148.318
C00772=1216.254,244.835,-61.410,-177.037,6.523,148.318
C00773=1216.259,244.586,-61.383,-177.039,6.521,148.319
C00774=1216.263,244.338,-61.357,-177.042,6.519,148.319
C00775=1216.268,244.089,-61.331,-177.044,6.517,148.319
C00776=1216.273,243.840,-61.305,-177.046,6.515,148.319
C00777=1216.277,243.592,-61.279,-177.049,6.513,148.320
C00778=1216.282,243.343,-61.252,-177.052,6.510,148.320
C00779=1216.286,243.094,-61.227,-177.055,6.508,148.320
C00780=1216.290,242.846,-61.200,-177.057,6.506,148.320
C00781=1216.295,242.597,-61.174,-177.060,6.504,148.321
C00782=1216.299,242.349,-61.149,-177.062,6.502,148.321
C00783=1216.303,242.101,-61.122,-177.064,6.500,148.321
C00784=1216.308,241.852,-61.096,-177.067,6.498,148.321
C00785=1216.313,241.603,-61.070,-177.070,6.496,148.322
C00786=1216.317,241.355,-61.043,-177.072,6.495,148.322
C00787=1216.322,241.106,-61.017,-177.074,6.492,148.322
C00788=1216.326,240.857,-60.992,-177.077,6.491,148.322
C00789=1216.331,240.609,-60.966,-177.080,6.488,148.323
C00790=1216.334,240.360,-60.940,-177.083,6.486,148.323
C00791=1216.339,240.111,-60.913,-177.085,6.484,148.323
C00792=1216.344,239.862,-60.887,-177.088,6.482,148.323
C00793=1216.348,239.614,-60.862,-177.090,6.480,148.324
C00794=1216.352,239.366,-60.836,-177.093,6.478,148.324
C00795=1216.357,239.117,-60.809,-177.095,6.476,148.324
C00796=1216.362,238.868,-60.783,-177.098,6.474,148.324
C00797=1216.366,238.620,-60.758,-177.100,6.472,148.325
C00798=1216.371,238.371,-60.732,-177.103,6.470,148.325
C00799=1216.376,238.122,-60.706,-177.105,6.468,148.325
C00800=1216.380,237.873,-60.680,-177.108,6.466,148.325
C00801=1216.385,237.603,-60.652,-177.111,6.464,148.326
C00802=1216.389,237.331,-60.624,-177.113,6.462,148.326
C00803=1216.394,237.060,-60.595,-177.116,6.460,148.326
C00804=1216.399,236.788,-60.567,-177.119,6.457,148.327
C00805=1216.403,236.540,-60.542,-177.121,6.455,148.327
C00806=1216.408,236.291,-60.515,-177.124,6.453,148.327
C00807=1216.413,236.042,-60.490,-177.127,6.451,148.327
C00808=1216.417,235.794,-60.464,-177.129,6.449,148.328
C00809=1216.422,235.545,-60.438,-177.132,6.448,148.328
C00810=1216.426,235.297,-60.413,-177.134,6.445,148.328
C00811=1216.431,235.048,-60.387,-177.137,6.444,148.328
C00812=1216.435,234.799,-60.362,-177.139,6.442,148.329
C00813=1216.439,234.550,-60.336,-177.142,6.440,148.329
C00814=1216.444,234.302,-60.310,-177.144,6.438,148.329
C00815=1216.449,234.053,-60.284,-177.147,6.436,148.329
C00816=1216.453,233.804,-60.258,-177.150,6.433,148.330
C00817=1216.458,233.556,-60.233,-177.152,6.431,148.330
C00818=1216.462,233.307,-60.207,-177.155,6.429,148.330
C00819=1216.466,233.059,-60.181,-177.157,6.427,148.330
C00820=1216.471,232.810,-60.156,-177.160,6.425,148.331
C00821=1216.475,232.562,-60.130,-177.162,6.424,148.331
C00822=1216.480,232.312,-60.105,-177.165,6.422,148.331
C00823=1216.485,232.064,-60.080,-177.168,6.420,148.332
C00824=1216.489,231.815,-60.054,-177.170,6.418,148.332
C00825=1216.493,231.567,-60.028,-177.172,6.416,148.332
C00826=1216.498,231.318,-60.003,-177.175,6.414,148.332
C00827=1216.502,231.070,-59.977,-177.178,6.412,148.333
C00828=1216.507,230.821,-59.953,-177.180,6.410,148.333
C00829=1216.512,230.572,-59.927,-177.182,6.408,148.333
C00830=1216.516,230.323,-59.901,-177.185,6.406,148.334
C00831=1216.521,230.075,-59.876,-177.188,6.404,148.334
C00832=1216.525,229.826,-59.850,-177.190,6.402,148.334
C00833=1216.529,229.577,-59.825,-177.193,6.401,148.335
C00834=1216.534,229.329,-59.799,-177.196,6.399,148.335
C00835=1216.539,229.080,-59.774,-177.198,6.397,148.335
C00836=1216.543,228.832,-59.748,-177.200,6.395,148.335
C00837=1216.548,228.583,-59.723,-177.203,6.393,148.336
C00838=1216.553,228.334,-59.698,-177.206,6.391,148.336
C00839=1216.556,228.086,-59.673,-177.208,6.389,148.336
C00840=1216.561,227.836,-59.648,-177.211,6.387,148.337
C00841=1216.566,227.588,-59.622,-177.213,6.385,148.337
C00842=1216.570,227.340,-59.597,-177.216,6.383,148.337
C00843=1216.575,227.091,-59.572,-177.218,6.381,148.337
C00844=1216.579,226.842,-59.546,-177.221,6.380,148.338
C00845=1216.584,226.594,-59.521,-177.224,6.378,148.338
C00846=1216.588,226.345,-59.496,-177.226,6.376,148.338
C00847=1216.592,226.096,-59.471,-177.228,6.374,148.338
C00848=1216.597,225.847,-59.446,-177.231,6.372,148.339
C00849=1216.601,225.599,-59.420,-177.234,6.370,148.339
C00850=1216.606,225.350,-59.395,-177.236,6.368,148.339
C00851=1216.611,225.101,-59.370,-177.239,6.366,148.340
C00852=1216.616,224.853,-59.344,-177.241,6.364,148.340
C00853=1216.619,224.604,-59.320,-177.244,6.363,148.340
C00854=1216.624,224.356,-59.295,-177.246,6.360,148.340
C00855=1216.629,224.106,-59.270,-177.249,6.359,148.341
C00856=1216.633,223.858,-59.244,-177.252,6.357,148.341
C00857=1216.638,223.609,-59.219,-177.254,6.355,148.341
C00858=1216.642,223.361,-59.194,-177.257,6.353,148.342
C00859=1216.647,223.111,-59.169,-177.259,6.351,148.342
C00860=1216.651,222.863,-59.144,-177.262,6.349,148.342
C00861=1216.656,222.614,-59.119,-177.265,6.347,148.343
C00862=1216.660,222.366,-59.095,-177.267,6.345,148.343
C00863=1216.665,222.117,-59.069,-177.269,6.343,148.343
C00864=1216.670,221.868,-59.044,-177.272,6.342,148.343
C00865=1216.674,221.619,-59.019,-177.275,6.340,148.344
C00866=1216.678,221.371,-58.995,-177.277,6.338,148.344
C00867=1216.683,221.123,-58.969,-177.280,6.336,148.344
C00868=1216.688,220.873,-58.944,-177.283,6.334,148.345
C00869=1216.692,220.625,-58.920,-177.285,6.332,148.345
C00870=1216.696,220.376,-58.894,-177.288,6.330,148.345
C00871=1216.701,220.127,-58.870,-177.291,6.329,148.346
C00872=1216.705,219.878,-58.845,-177.293,6.326,148.346
C00873=1216.710,219.630,-58.820,-177.295,6.325,148.346
C00874=1216.715,219.381,-58.795,-177.298,6.323,148.347
C00875=1216.719,219.132,-58.771,-177.301,6.321,148.347
C00876=1216.724,218.884,-58.746,-177.303,6.319,148.347
C00877=1216.728,218.635,-58.720,-177.306,6.317,148.348
C00878=1216.733,218.386,-58.696,-177.308,6.315,148.348
C00879=1216.737,218.137,-58.671,-177.311,6.313,148.348
C00880=1216.742,217.889,-58.647,-177.314,6.312,148.349
C00881=1216.747,217.640,-58.622,-177.316,6.310,148.349
C00882=1216.751,217.391,-58.597,-177.319,6.308,148.349
C00883=1216.755,217.143,-58.573,-177.322,6.306,148.350
C00884=1216.760,216.893,-58.548,-177.324,6.304,148.350
C00885=1216.764,216.645,-58.523,-177.326,6.302,148.350
C00886=1216.769,216.397,-58.498,-177.329,6.300,148.350
C00887=1216.774,216.147,-58.473,-177.332,6.298,148.351
C00888=1216.778,215.899,-58.449,-177.334,6.296,148.351
C00889=1216.783,215.650,-58.424,-177.337,6.295,148.351
C00890=1216.787,215.401,-58.400,-177.340,6.293,148.352
C00891=1216.792,215.152,-58.375,-177.342,6.291,148.352
C00892=1216.797,214.904,-58.351,-177.345,6.289,148.352
C00893=1216.801,214.655,-58.325,-177.348,6.287,148.353
C00894=1216.805,214.407,-58.301,-177.350,6.285,148.353
C00895=1216.810,214.158,-58.277,-177.353,6.284,148.353
C00896=1216.814,213.909,-58.252,-177.355,6.282,148.354
C00897=1216.819,213.660,-58.228,-177.358,6.280,148.354
C00898=1216.824,213.412,-58.203,-177.360,6.279,148.354
C00899=1216.828,213.162,-58.178,-177.363,6.277,148.355
C00900=1216.833,212.914,-58.154,-177.365,6.275,148.355
C00901=1216.838,212.665,-58.130,-177.368,6.273,148.355
C00902=1216.841,212.416,-58.105,-177.370,6.271,148.355
C00903=1216.846,212.168,-58.081,-177.373,6.269,148.356
C00904=1216.851,211.919,-58.056,-177.375,6.267,148.356
C00905=1216.856,211.649,-58.030,-177.379,6.266,148.357
C00906=1216.861,211.377,-58.003,-177.382,6.263,148.357
C00907=1216.865,211.107,-57.977,-177.384,6.261,148.357
C00908=1216.871,210.837,-57.951,-177.387,6.260,148.358
C00909=1216.876,210.588,-57.926,-177.390,6.258,148.358
C00910=1216.880,210.340,-57.902,-177.392,6.256,148.358
C00911=1216.884,210.091,-57.877,-177.395,6.254,148.359
C00912=1216.889,209.842,-57.853,-177.398,6.252,148.359
C00913=1216.894,209.593,-57.829,-177.400,6.250,148.359
C00914=1216.898,209.345,-57.805,-177.402,6.249,148.360
C00915=1216.903,209.095,-57.780,-177.405,6.247,148.360
C00916=1216.907,208.847,-57.756,-177.408,6.246,148.360
C00917=1216.911,208.598,-57.732,-177.410,6.244,148.361
C00918=1216.917,208.350,-57.707,-177.413,6.242,148.361
C00919=1216.921,208.100,-57.684,-177.416,6.240,148.361
C00920=1216.925,207.852,-57.660,-177.418,6.238,148.362
C00921=1216.930,207.603,-57.635,-177.421,6.236,148.362
C00922=1216.935,207.354,-57.611,-177.423,6.235,148.362
C00923=1216.939,207.106,-57.587,-177.426,6.233,148.363
C00924=1216.944,206.856,-57.562,-177.429,6.231,148.363
C00925=1216.948,206.608,-57.538,-177.431,6.229,148.363
C00926=1216.953,206.359,-57.514,-177.433,6.228,148.364
C00927=1216.958,206.110,-57.490,-177.436,6.226,148.364
C00928=1216.962,205.861,-57.466,-177.439,6.224,148.364
C00929=1216.967,205.613,-57.442,-177.441,6.222,148.365
C00930=1216.971,205.364,-57.418,-177.444,6.221,148.365
C00931=1216.975,205.115,-57.394,-177.447,6.219,148.365
C00932=1216.980,204.866,-57.370,-177.449,6.217,148.366
C00933=1216.985,204.618,-57.346,-177.452,6.215,148.366
C00934=1216.990,204.369,-57.322,-177.455,6.213,148.366
C00935=1216.994,204.120,-57.298,-177.457,6.212,148.367
C00936=1216.998,203.871,-57.273,-177.459,6.210,148.367
C00937=1217.003,203.622,-57.250,-177.462,6.209,148.368
C00938=1217.008,203.373,-57.226,-177.465,6.207,148.368
C00939=1217.012,203.124,-57.202,-177.467,6.205,148.368
C00940=1217.017,202.876,-57.178,-177.470,6.203,148.369
C00941=1217.021,202.628,-57.154,-177.473,6.201,148.369
C00942=1217.027,202.378,-57.130,-177.475,6.199,148.369
C00943=1217.031,202.130,-57.106,-177.478,6.198,148.370
C00944=1217.035,201.880,-57.083,-177.480,6.197,148.370
C00945=1217.039,201.632,-57.058,-177.483,6.195,148.370
C00946=1217.044,201.383,-57.035,-177.485,6.193,148.371
C00947=1217.048,201.134,-57.011,-177.488,6.191,148.371
C00948=1217.053,200.885,-56.988,-177.490,6.189,148.371
C00949=1217.058,200.637,-56.964,-177.493,6.187,148.372
C00950=1217.063,200.387,-56.940,-177.496,6.185,148.372
C00951=1217.067,200.139,-56.916,-177.498,6.184,148.372
C00952=1217.072,199.890,-56.892,-177.500,6.183,148.373
C00953=1217.077,199.642,-56.868,-177.503,6.181,148.373
C00954=1217.081,199.393,-56.845,-177.506,6.179,148.373
C00955=1217.086,199.143,-56.821,-177.508,6.177,148.374
C00956=1217.090,198.895,-56.797,-177.511,6.175,148.374
C00957=1217.094,198.645,-56.774,-177.514,6.173,148.374
C00958=1217.099,198.397,-56.750,-177.516,6.173,148.375
C00959=1217.103,198.148,-56.726,-177.519,6.171,148.375
C00960=1217.108,197.899,-56.703,-177.522,6.169,148.376
C00961=1217.113,197.650,-56.679,-177.524,6.167,148.376
C00962=1217.117,197.401,-56.655,-177.527,6.165,148.376
C00963=1217.122,197.152,-56.632,-177.529,6.164,148.377
C00964=1217.126,196.904,-56.608,-177.532,6.162,148.377
C00965=1217.131,196.655,-56.585,-177.534,6.161,148.377
C00966=1217.136,196.406,-56.561,-177.537,6.159,148.378
C00967=1217.140,196.158,-56.537,-177.539,6.157,148.378
C00968=1217.145,195.908,-56.514,-177.542,6.155,148.378
C00969=1217.150,195.659,-56.490,-177.545,6.153,148.379
C00970=1217.154,195.410,-56.467,-177.547,6.152,148.379
C00971=1217.159,195.162,-56.443,-177.550,6.151,148.380
C00972=1217.163,194.913,-56.420,-177.552,6.149,148.380
C00973=1217.168,194.664,-56.396,-177.555,6.147,148.380
C00974=1217.173,194.415,-56.373,-177.558,6.145,148.381
C00975=1217.177,194.166,-56.349,-177.561,6.144,148.381
C00976=1217.182,193.917,-56.326,-177.563,6.143,148.382
C00977=1217.187,193.668,-56.302,-177.565,6.141,148.382
C00978=1217.191,193.420,-56.280,-177.568,6.139,148.382
C00979=1217.196,193.171,-56.256,-177.571,6.137,148.383
C00980=1217.201,192.922,-56.233,-177.573,6.135,148.383
C00981=1217.205,192.674,-56.209,-177.576,6.133,148.383
C00982=1217.210,192.425,-56.186,-177.578,6.132,148.384
C00983=1217.214,192.176,-56.162,-177.581,6.131,148.384
C00984=1217.219,191.927,-56.139,-177.583,6.129,148.384
C00985=1217.224,191.678,-56.116,-177.586,6.127,148.385
C00986=1217.228,191.429,-56.093,-177.589,6.125,148.385
C00987=1217.232,191.180,-56.069,-177.591,6.124,148.386
C00988=1217.237,190.931,-56.046,-177.594,6.123,148.386
C00989=1217.242,190.682,-56.023,-177.596,6.121,148.386
C00990=1217.246,190.433,-55.999,-177.599,6.119,148.387
C00991=1217.252,190.185,-55.976,-177.602,6.117,148.387
C00992=1217.255,189.937,-55.953,-177.604,6.116,148.387
C00993=1217.260,189.687,-55.929,-177.606,6.114,148.388
C00994=1217.265,189.438,-55.906,-177.609,6.112,148.388
C00995=1217.270,189.189,-55.883,-177.612,6.111,148.388
C00996=1217.274,188.940,-55.859,-177.615,6.109,148.389
C00997=1217.279,188.691,-55.837,-177.617,6.108,148.389
C00998=1217.283,188.442,-55.814,-177.620,6.106,148.390
C00999=1217.289,188.194,-55.791,-177.622,6.104,148.390
C01000=1217.293,187.945,-55.768,-177.625,6.103,148.390
C01001=1217.297,187.696,-55.745,-177.627,6.102,148.391
C01002=1217.302,187.447,-55.722,-177.630,6.100,148.391
C01003=1217.307,187.198,-55.698,-177.632,6.098,148.392
C01004=1217.311,186.949,-55.675,-177.635,6.096,148.392
C01005=1217.315,186.700,-55.652,-177.638,6.095,148.392
C01006=1217.321,186.452,-55.629,-177.640,6.094,148.393
C01007=1217.325,186.203,-55.606,-177.643,6.092,148.393
C01008=1217.329,185.954,-55.583,-177.646,6.090,148.394
C01009=1217.335,185.684,-55.558,-177.648,6.088,148.394
C01010=1217.340,185.414,-55.533,-177.651,6.087,148.394
C01011=1217.344,185.145,-55.508,-177.654,6.085,148.395
C01012=1217.350,184.875,-55.483,-177.657,6.083,148.395
C01013=1217.354,184.627,-55.461,-177.659,6.081,148.396
C01014=1217.359,184.377,-55.438,-177.662,6.080,148.396
C01015=1217.363,184.128,-55.415,-177.665,6.079,148.396
C01016=1217.368,183.880,-55.392,-177.667,6.077,148.397
C01017=1217.373,183.631,-55.369,-177.670,6.075,148.397
C01018=1217.377,183.382,-55.346,-177.672,6.074,148.398
C01019=1217.382,183.132,-55.323,-177.675,6.072,148.398
C01020=1217.387,182.884,-55.300,-177.677,6.070,148.398
C01021=1217.391,182.635,-55.278,-177.680,6.069,148.399
C01022=1217.396,182.386,-55.255,-177.682,6.068,148.399
C01023=1217.401,182.137,-55.232,-177.685,6.066,148.400
C01024=1217.405,181.889,-55.209,-177.688,6.064,148.400
C01025=1217.410,181.640,-55.186,-177.690,6.062,148.400
C01026=1217.414,181.390,-55.164,-177.692,6.061,148.401
C01027=1217.419,181.141,-55.141,-177.696,6.060,148.401
C01028=1217.423,180.893,-55.118,-177.698,6.058,148.402
C01029=1217.428,180.644,-55.095,-177.701,6.056,148.402
C01030=1217.432,180.395,-55.073,-177.703,6.055,148.402
C01031=1217.437,180.145,-55.050,-177.706,6.053,148.403
C01032=1217.442,179.897,-55.028,-177.708,6.052,148.403
C01033=1217.447,179.648,-55.004,-177.711,6.051,148.404
C01034=1217.451,179.399,-54.982,-177.714,6.049,148.404
C01035=1217.456,179.151,-54.959,-177.716,6.047,148.404
C01036=1217.460,178.901,-54.937,-177.719,6.045,148.405
C01037=1217.465,178.652,-54.914,-177.721,6.044,148.405
C01038=1217.469,178.403,-54.892,-177.724,6.043,148.405
C01039=1217.475,178.154,-54.869,-177.727,6.041,148.406
C01040=1217.479,177.906,-54.846,-177.729,6.040,148.406
C01041=1217.484,177.656,-54.823,-177.732,6.038,148.407
C01042=1217.488,177.408,-54.801,-177.734,6.036,148.407
C01043=1217.493,177.158,-54.778,-177.737,6.035,148.408
C01044=1217.497,176.910,-54.756,-177.739,6.034,148.408
C01045=1217.503,176.661,-54.733,-177.742,6.032,148.408
C01046=1217.507,176.411,-54.711,-177.745,6.030,148.409
C01047=1217.511,176.163,-54.689,-177.747,6.029,148.409
C01048=1217.517,175.914,-54.666,-177.749,6.027,148.410
C01049=1217.521,175.665,-54.643,-177.752,6.026,148.410
C01050=1217.526,175.416,-54.621,-177.755,6.024,148.411
C01051=1217.530,175.167,-54.598,-177.757,6.023,148.411
C01052=1217.534,174.918,-54.576,-177.760,6.021,148.411
C01053=1217.540,174.669,-54.554,-177.763,6.020,148.412
C01054=1217.544,174.420,-54.531,-177.765,6.019,148.412
C01055=1217.548,174.171,-54.509,-177.768,6.017,148.413
C01056=1217.554,173.923,-54.486,-177.771,6.015,148.413
C01057=1217.558,173.673,-54.464,-177.773,6.014,148.413
C01058=1217.563,173.425,-54.443,-177.775,6.012,148.414
C01059=1217.567,173.176,-54.419,-177.778,6.011,148.414
C01060=1217.572,172.926,-54.397,-177.781,6.010,148.415
C01061=1217.577,172.678,-54.376,-177.783,6.008,148.415
C01062=1217.582,172.428,-54.353,-177.786,6.006,148.415
C01063=1217.586,172.180,-54.330,-177.788,6.005,148.416
C01064=1217.590,171.931,-54.308,-177.791,6.004,148.416
C01065=1217.595,171.681,-54.286,-177.794,6.002,148.417
C01066=1217.600,171.433,-54.263,-177.796,6.001,148.417
C01067=1217.604,171.184,-54.241,-177.799,5.999,148.417
C01068=1217.609,170.935,-54.220,-177.801,5.997,148.418
C01069=1217.614,170.685,-54.197,-177.804,5.996,148.418
C01070=1217.619,170.437,-54.175,-177.806,5.995,148.419
C01071=1217.623,170.188,-54.153,-177.809,5.993,148.419
C01072=1217.628,169.939,-54.131,-177.811,5.992,148.420
C01073=1217.633,169.690,-54.108,-177.814,5.991,148.420
C01074=1217.638,169.441,-54.087,-177.817,5.989,148.421
C01075=1217.642,169.192,-54.064,-177.819,5.988,148.421
C01076=1217.647,168.944,-54.042,-177.822,5.986,148.421
C01077=1217.652,168.694,-54.019,-177.825,5.984,148.422
C01078=1217.656,168.445,-53.997,-177.827,5.983,148.422
C01079=1217.661,168.196,-53.976,-177.830,5.982,148.423
C01080=1217.665,167.947,-53.954,-177.832,5.980,148.423
C01081=1217.670,167.698,-53.932,-177.834,5.979,148.423
C01082=1217.675,167.448,-53.909,-177.838,5.977,148.424
C01083=1217.680,167.200,-53.888,-177.840,5.976,148.424
C01084=1217.684,166.950,-53.866,-177.842,5.975,148.425
C01085=1217.689,166.702,-53.844,-177.845,5.973,148.425
C01086=1217.693,166.454,-53.822,-177.848,5.971,148.426
C01087=1217.698,166.204,-53.799,-177.850,5.970,148.426
C01088=1217.703,165.956,-53.778,-177.853,5.968,148.426
C01089=1217.708,165.706,-53.755,-177.856,5.967,148.427
C01090=1217.712,165.457,-53.733,-177.858,5.966,148.427
C01091=1217.717,165.208,-53.711,-177.861,5.964,148.428
C01092=1217.722,164.960,-53.690,-177.863,5.963,148.428
C01093=1217.726,164.710,-53.668,-177.866,5.962,148.429
C01094=1217.731,164.462,-53.646,-177.869,5.960,148.429
C01095=1217.735,164.212,-53.624,-177.871,5.959,148.429
C01096=1217.740,163.964,-53.602,-177.873,5.957,148.430
C01097=1217.744,163.714,-53.581,-177.877,5.956,148.430
C01098=1217.749,163.465,-53.559,-177.879,5.955,148.431
C01099=1217.754,163.216,-53.538,-177.881,5.953,148.431
C01100=1217.758,162.967,-53.516,-177.883,5.952,148.432
C01101=1217.763,162.718,-53.494,-177.887,5.950,148.432
C01102=1217.768,162.469,-53.472,-177.889,5.949,148.433
C01103=1217.772,162.220,-53.450,-177.891,5.948,148.433
C01104=1217.777,161.972,-53.428,-177.895,5.946,148.434
C01105=1217.782,161.722,-53.406,-177.897,5.944,148.434
C01106=1217.786,161.474,-53.385,-177.899,5.943,148.434
C01107=1217.791,161.224,-53.363,-177.902,5.941,148.435
C01108=1217.796,160.975,-53.342,-177.905,5.941,148.435
C01109=1217.801,160.726,-53.320,-177.907,5.939,148.436
C01110=1217.805,160.477,-53.298,-177.910,5.937,148.436
C01111=1217.810,160.229,-53.276,-177.912,5.937,148.437
C01112=1217.814,159.979,-53.255,-177.915,5.935,148.437
C01113=1217.820,159.710,-53.231,-177.918,5.933,148.437
C01114=1217.825,159.440,-53.208,-177.920,5.932,148.438
C01115=1217.830,159.171,-53.185,-177.923,5.930,148.438
C01116=1217.835,158.903,-53.161,-177.926,5.929,148.439
C01117=1217.840,158.653,-53.140,-177.929,5.927,148.439
C01118=1217.845,158.405,-53.118,-177.931,5.926,148.440
C01119=1217.849,158.156,-53.097,-177.934,5.925,148.440
C01120=1217.853,157.907,-53.075,-177.936,5.924,148.441
C01121=1217.859,157.658,-53.054,-177.939,5.922,148.441
C01122=1217.863,157.408,-53.032,-177.942,5.921,148.442
C01123=1217.868,157.160,-53.010,-177.944,5.919,148.442
C01124=1217.873,156.911,-52.989,-177.947,5.918,148.442
C01125=1217.877,156.661,-52.967,-177.949,5.917,148.443
C01126=1217.882,156.413,-52.946,-177.952,5.915,148.443
C01127=1217.887,156.163,-52.925,-177.954,5.914,148.444
C01128=1217.891,155.915,-52.903,-177.957,5.912,148.444
C01129=1217.896,155.666,-52.881,-177.960,5.911,148.445
C01130=1217.901,155.416,-52.860,-177.962,5.910,148.445
C01131=1217.906,155.168,-52.839,-177.965,5.908,148.446
C01132=1217.910,154.918,-52.817,-177.967,5.907,148.446
C01133=1217.915,154.669,-52.796,-177.970,5.906,148.447
C01134=1217.919,154.421,-52.775,-177.972,5.905,148.447
C01135=1217.924,154.172,-52.754,-177.975,5.903,148.448
C01136=1217.929,153.922,-52.732,-177.977,5.902,148.448
C01137=1217.934,153.673,-52.711,-177.980,5.900,148.448
C01138=1217.939,153.424,-52.689,-177.983,5.899,148.449
C01139=1217.943,153.175,-52.669,-177.985,5.898,148.449
C01140=1217.947,152.926,-52.647,-177.988,5.896,148.450
C01141=1217.953,152.677,-52.626,-177.991,5.896,148.450
C01142=1217.958,152.428,-52.604,-177.993,5.894,148.451
C01143=1217.963,152.179,-52.583,-177.995,5.893,148.451
C01144=1217.966,151.930,-52.562,-177.999,5.891,148.452
C01145=1217.971,151.681,-52.541,-178.001,5.890,148.452
C01146=1217.976,151.432,-52.519,-178.003,5.888,148.452
C01147=1217.981,151.183,-52.498,-178.006,5.887,148.453
C01148=1217.985,150.933,-52.477,-178.009,5.886,148.453
C01149=1217.990,150.684,-52.455,-178.011,5.884,148.454
C01150=1217.995,150.435,-52.434,-178.014,5.884,148.454
C01151=1217.999,150.187,-52.413,-178.017,5.882,148.455
C01152=1218.005,149.938,-52.392,-178.019,5.881,148.455
C01153=1218.009,149.688,-52.371,-178.022,5.879,148.456
C01154=1218.013,149.439,-52.350,-178.024,5.878,148.456
C01155=1218.019,149.190,-52.329,-178.027,5.877,148.457
C01156=1218.024,148.941,-52.308,-178.029,5.876,148.457
C01157=1218.028,148.692,-52.287,-178.032,5.874,148.458
C01158=1218.033,148.443,-52.266,-178.034,5.873,148.458
C01159=1218.038,148.193,-52.245,-178.037,5.872,148.459
C01160=1218.042,147.945,-52.224,-178.040,5.870,148.459
C01161=1218.047,147.696,-52.203,-178.042,5.869,148.460
C01162=1218.052,147.446,-52.182,-178.045,5.867,148.460
C01163=1218.056,147.198,-52.161,-178.047,5.866,148.460
C01164=1218.061,146.949,-52.140,-178.050,5.865,148.461
C01165=1218.065,146.699,-52.119,-178.052,5.864,148.461
C01166=1218.070,146.450,-52.098,-178.056,5.863,148.462
C01167=1218.075,146.201,-52.076,-178.058,5.862,148.462
C01168=1218.080,145.952,-52.056,-178.060,5.860,148.463
C01169=1218.085,145.703,-52.035,-178.063,5.859,148.463
C01170=1218.089,145.454,-52.015,-178.066,5.857,148.464
C01171=1218.094,145.205,-51.993,-178.068,5.856,148.464
C01172=1218.099,144.956,-51.972,-178.071,5.855,148.465
C01173=1218.103,144.706,-51.951,-178.073,5.854,148.465
C01174=1218.108,144.457,-51.930,-178.076,5.852,148.466
C01175=1218.113,144.208,-51.910,-178.078,5.851,148.466
C01176=1218.118,143.959,-51.889,-178.081,5.850,148.466
C01177=1218.122,143.711,-51.868,-178.084,5.849,148.467
C01178=1218.127,143.461,-51.847,-178.086,5.847,148.467
C01179=1218.132,143.213,-51.826,-178.089,5.847,148.468
C01180=1218.137,142.963,-51.805,-178.091,5.845,148.468
C01181=1218.141,142.714,-51.785,-178.094,5.844,148.469
C01182=1218.146,142.465,-51.764,-178.097,5.842,148.470
C01183=1218.151,142.216,-51.744,-178.099,5.841,148.470
C01184=1218.156,141.967,-51.723,-178.102,5.840,148.470
C01185=1218.160,141.717,-51.702,-178.104,5.839,148.471
C01186=1218.165,141.468,-51.681,-178.107,5.837,148.471
C01187=1218.169,141.220,-51.660,-178.109,5.837,148.472
C01188=1218.174,140.971,-51.640,-178.112,5.835,148.472
C01189=1218.179,140.721,-51.619,-178.115,5.834,148.473
C01190=1218.183,140.472,-51.598,-178.117,5.832,148.473
C01191=1218.188,140.223,-51.577,-178.119,5.831,148.474
C01192=1218.193,139.974,-51.557,-178.122,5.831,148.474
C01193=1218.198,139.725,-51.536,-178.125,5.829,148.475
C01194=1218.203,139.476,-51.516,-178.127,5.828,148.475
C01195=1218.207,139.227,-51.495,-178.130,5.826,148.476
C01196=1218.212,138.978,-51.474,-178.132,5.825,148.476
C01197=1218.217,138.728,-51.455,-178.135,5.824,148.477
C01198=1218.222,138.479,-51.434,-178.137,5.823,148.477
C01199=1218.226,138.230,-51.413,-178.141,5.822,148.478
C01200=1218.231,137.981,-51.393,-178.143,5.821,148.478
C01201=1218.236,137.732,-51.372,-178.145,5.819,148.479
C01202=1218.241,137.483,-51.352,-178.148,5.818,148.479
C01203=1218.245,137.234,-51.331,-178.151,5.816,148.480
C01204=1218.250,136.985,-51.310,-178.153,5.816,148.480
C01205=1218.255,136.736,-51.290,-178.156,5.814,148.481
C01206=1218.259,136.487,-51.269,-178.158,5.813,148.481
C01207=1218.264,136.237,-51.249,-178.161,5.812,148.482
C01208=1218.269,135.988,-51.229,-178.163,5.811,148.482
C01209=1218.273,135.739,-51.208,-178.166,5.810,148.483
C01210=1218.279,135.490,-51.187,-178.169,5.808,148.483
C01211=1218.283,135.241,-51.167,-178.171,5.808,148.484
C01212=1218.287,134.992,-51.147,-178.174,5.806,148.484
C01213=1218.293,134.743,-51.127,-178.176,5.805,148.485
C01214=1218.298,134.494,-51.106,-178.179,5.803,148.485
C01215=1218.302,134.245,-51.086,-178.182,5.803,148.486
C01216=1218.307,133.996,-51.066,-178.184,5.802,148.486
C01217=1218.312,133.727,-51.044,-178.187,5.800,148.487
C01218=1218.317,133.458,-51.021,-178.190,5.798,148.487
C01219=1218.322,133.189,-51.000,-178.192,5.798,148.488
C01220=1218.327,132.921,-50.978,-178.195,5.796,148.488
C01221=1218.332,132.671,-50.958,-178.198,5.795,148.489
C01222=1218.337,132.422,-50.938,-178.200,5.794,148.489
C01223=1218.342,132.173,-50.917,-178.203,5.793,148.490
C01224=1218.347,131.923,-50.897,-178.206,5.791,148.490
C01225=1218.352,131.675,-50.877,-178.208,5.791,148.491
C01226=1218.356,131.426,-50.857,-178.210,5.790,148.491
C01227=1218.361,131.177,-50.837,-178.213,5.788,148.492
C01228=1218.366,130.927,-50.816,-178.216,5.787,148.492
C01229=1218.370,130.678,-50.796,-178.219,5.786,148.493
C01230=1218.375,130.429,-50.776,-178.221,5.785,148.493
C01231=1218.380,130.180,-50.756,-178.224,5.783,148.494
C01232=1218.384,129.931,-50.735,-178.226,5.782,148.494
C01233=1218.390,129.682,-50.716,-178.229,5.782,148.495
C01234=1218.395,129.433,-50.695,-178.231,5.780,148.495
C01235=1218.399,129.183,-50.675,-178.233,5.779,148.496
C01236=1218.404,128.934,-50.655,-178.237,5.777,148.496
C01237=1218.408,128.685,-50.635,-178.239,5.777,148.497
C01238=1218.413,128.436,-50.615,-178.241,5.776,148.497
C01239=1218.418,128.188,-50.595,-178.244,5.774,148.498
C01240=1218.423,127.938,-50.575,-178.247,5.773,148.498
C01241=1218.427,127.689,-50.555,-178.249,5.772,148.499
C01242=1218.433,127.439,-50.535,-178.252,5.771,148.499
C01243=1218.437,127.190,-50.514,-178.254,5.770,148.500
C01244=1218.442,126.941,-50.495,-178.257,5.769,148.500
C01245=1218.447,126.692,-50.475,-178.259,5.768,148.501
C01246=1218.452,126.443,-50.455,-178.263,5.766,148.501
C01247=1218.456,126.194,-50.435,-178.265,5.765,148.502
C01248=1218.461,125.944,-50.415,-178.267,5.765,148.502
C01249=1218.465,125.695,-50.395,-178.270,5.763,148.503
C01250=1218.471,125.447,-50.375,-178.273,5.762,148.503
C01251=1218.475,125.197,-50.356,-178.275,5.760,148.504
C01252=1218.480,124.948,-50.335,-178.278,5.760,148.504
C01253=1218.484,124.698,-50.316,-178.280,5.759,148.505
C01254=1218.489,124.450,-50.296,-178.283,5.757,148.505
C01255=1218.494,124.201,-50.276,-178.285,5.756,148.506
C01256=1218.499,123.951,-50.256,-178.288,5.755,148.507
C01257=1218.503,123.702,-50.236,-178.290,5.754,148.507
C01258=1218.508,123.453,-50.216,-178.293,5.753,148.508
C01259=1218.513,123.204,-50.197,-178.296,5.752,148.508
C01260=1218.518,122.955,-50.177,-178.298,5.751,148.509
C01261=1218.523,122.705,-50.157,-178.301,5.750,148.509
C01262=1218.528,122.456,-50.138,-178.304,5.749,148.510
C01263=1218.532,122.207,-50.117,-178.306,5.748,148.510
C01264=1218.537,121.958,-50.098,-178.308,5.747,148.511
C01265=1218.542,121.708,-50.078,-178.311,5.745,148.511
C01266=1218.547,121.460,-50.058,-178.314,5.745,148.512
C01267=1218.552,121.210,-50.038,-178.316,5.743,148.512
C01268=1218.556,120.961,-50.019,-178.319,5.742,148.513
C01269=1218.561,120.711,-49.999,-178.321,5.741,148.513
C01270=1218.566,120.463,-49.979,-178.324,5.740,148.514
C01271=1218.570,120.214,-49.960,-178.326,5.739,148.514
C01272=1218.575,119.964,-49.940,-178.329,5.738,148.515
C01273=1218.580,119.715,-49.921,-178.332,5.736,148.515
C01274=1218.585,119.466,-49.901,-178.334,5.736,148.516
C01275=1218.590,119.217,-49.881,-178.336,5.735,148.516
C01276=1218.595,118.968,-49.862,-178.340,5.733,148.517
C01277=1218.600,118.718,-49.842,-178.342,5.733,148.517
C01278=1218.604,118.469,-49.822,-178.344,5.732,148.518
C01279=1218.609,118.221,-49.803,-178.348,5.730,148.519
C01280=1218.613,117.971,-49.783,-178.350,5.729,148.519
C01281=1218.618,117.722,-49.764,-178.352,5.729,148.520
C01282=1218.623,117.473,-49.744,-178.355,5.727,148.520
C01283=1218.628,117.223,-49.725,-178.358,5.726,148.521
C01284=1218.633,116.974,-49.705,-178.360,5.725,148.521
C01285=1218.638,116.725,-49.686,-178.363,5.724,148.522
C01286=1218.642,116.476,-49.667,-178.365,5.723,148.522
C01287=1218.647,116.227,-49.646,-178.368,5.722,148.523
C01288=1218.652,115.978,-49.627,-178.370,5.721,148.523
C01289=1218.657,115.728,-49.607,-178.373,5.720,148.524
C01290=1218.661,115.480,-49.589,-178.376,5.719,148.524
C01291=1218.666,115.230,-49.569,-178.378,5.718,148.525
C01292=1218.671,114.981,-49.549,-178.381,5.717,148.525
C01293=1218.676,114.732,-49.530,-178.383,5.716,148.526
C01294=1218.681,114.482,-49.511,-178.386,5.715,148.526
C01295=1218.686,114.234,-49.492,-178.388,5.714,148.527
C01296=1218.690,113.984,-49.472,-178.391,5.713,148.528
C01297=1218.695,113.734,-49.453,-178.393,5.711,148.528
C01298=1218.700,113.486,-49.433,-178.396,5.711,148.529
C01299=1218.704,113.236,-49.414,-178.399,5.710,148.529
C01300=1218.710,112.987,-49.395,-178.401,5.708,148.530
C01301=1218.715,112.738,-49.375,-178.404,5.708,148.530
C01302=1218.719,112.489,-49.357,-178.406,5.707,148.531
C01303=1218.724,112.240,-49.337,-178.409,5.705,148.531
C01304=1218.729,111.990,-49.317,-178.411,5.704,148.532
C01305=1218.734,111.741,-49.299,-178.414,5.704,148.532
C01306=1218.738,111.491,-49.280,-178.417,5.702,148.533
C01307=1218.744,111.243,-49.260,-178.419,5.701,148.533
C01308=1218.748,110.993,-49.241,-178.422,5.701,148.534
C01309=1218.753,110.744,-49.222,-178.424,5.700,148.534
C01310=1218.758,110.495,-49.202,-178.427,5.698,148.535
C01311=1218.762,110.246,-49.184,-178.429,5.697,148.535
C01312=1218.767,109.997,-49.164,-178.432,5.697,148.536
C01313=1218.772,109.747,-49.144,-178.435,5.695,148.536
C01314=1218.777,109.498,-49.126,-178.437,5.694,148.537
C01315=1218.781,109.248,-49.107,-178.440,5.694,148.538
C01316=1218.787,109.000,-49.087,-178.443,5.692,148.538
C01317=1218.791,108.750,-49.068,-178.445,5.691,148.539
C01318=1218.796,108.501,-49.049,-178.447,5.691,148.539
C01319=1218.800,108.252,-49.031,-178.450,5.690,148.540
C01320=1218.806,108.003,-49.011,-178.453,5.688,148.541
C01321=1218.811,107.734,-48.990,-178.455,5.688,148.541
C01322=1218.817,107.465,-48.970,-178.458,5.686,148.542
C01323=1218.821,107.197,-48.950,-178.461,5.685,148.542
C01324=1218.826,106.929,-48.929,-178.464,5.684,148.543
C01325=1218.832,106.680,-48.910,-178.466,5.683,148.543
C01326=1218.836,106.430,-48.891,-178.469,5.682,148.544
C01327=1218.841,106.182,-48.872,-178.471,5.682,148.544
C01328=1218.845,105.932,-48.853,-178.474,5.680,148.545
C01329=1218.851,105.683,-48.834,-178.477,5.680,148.546
C01330=1218.855,105.434,-48.815,-178.479,5.679,148.546
C01331=1218.860,105.185,-48.796,-178.482,5.678,148.547
C01332=1218.865,104.935,-48.778,-178.484,5.676,148.547
C01333=1218.870,104.686,-48.759,-178.487,5.676,148.548
C01334=1218.874,104.437,-48.739,-178.490,5.675,148.548
C01335=1218.880,104.187,-48.721,-178.492,5.673,148.549
C01336=1218.884,103.939,-48.702,-178.495,5.673,148.549
C01337=1218.889,103.689,-48.683,-178.497,5.672,148.550
C01338=1218.894,103.440,-48.665,-178.500,5.671,148.550
C01339=1218.899,103.190,-48.645,-178.503,5.670,148.551
C01340=1218.903,102.941,-48.627,-178.505,5.669,148.551
C01341=1218.908,102.692,-48.607,-178.508,5.668,148.552
C01342=1218.913,102.443,-48.589,-178.510,5.667,148.553
C01343=1218.918,102.194,-48.570,-178.513,5.666,148.553
C01344=1218.922,101.944,-48.551,-178.515,5.665,148.554
C01345=1218.928,101.695,-48.532,-178.518,5.664,148.554
C01346=1218.932,101.446,-48.513,-178.520,5.664,148.555
C01347=1218.937,101.196,-48.495,-178.523,5.662,148.556
C01348=1218.942,100.948,-48.476,-178.525,5.661,148.556
C01349=1218.947,100.698,-48.458,-178.528,5.661,148.557
C01350=1218.952,100.449,-48.438,-178.530,5.660,148.557
C01351=1218.957,100.200,-48.420,-178.533,5.658,148.558
C01352=1218.961,99.950,-48.401,-178.536,5.658,148.558
C01353=1218.967,99.701,-48.383,-178.538,5.657,148.559
C01354=1218.971,99.452,-48.364,-178.541,5.656,148.559
C01355=1218.976,99.202,-48.345,-178.544,5.655,148.560
C01356=1218.981,98.954,-48.326,-178.546,5.654,148.560
C01357=1218.985,98.704,-48.308,-178.549,5.653,148.561
C01358=1218.991,98.455,-48.289,-178.551,5.652,148.562
C01359=1218.995,98.206,-48.271,-178.553,5.652,148.562
C01360=1219.000,97.956,-48.252,-178.557,5.650,148.563
C01361=1219.005,97.707,-48.233,-178.559,5.649,148.563
C01362=1219.010,97.458,-48.215,-178.561,5.649,148.564
C01363=1219.014,97.208,-48.196,-178.564,5.648,148.564
C01364=1219.020,96.959,-48.178,-178.567,5.646,148.565
C01365=1219.025,96.710,-48.160,-178.569,5.646,148.566
C01366=1219.029,96.461,-48.141,-178.572,5.645,148.566
C01367=1219.033,96.211,-48.123,-178.574,5.644,148.567
C01368=1219.039,95.962,-48.104,-178.577,5.643,148.567
C01369=1219.044,95.713,-48.085,-178.580,5.642,148.568
C01370=1219.048,95.463,-48.067,-178.582,5.641,148.568
C01371=1219.054,95.214,-48.048,-178.585,5.640,148.569
C01372=1219.058,94.965,-48.030,-178.587,5.640,148.570
C01373=1219.063,94.716,-48.011,-178.590,5.638,148.570
C01374=1219.068,94.466,-47.993,-178.593,5.638,148.571
C01375=1219.073,94.217,-47.975,-178.595,5.637,148.571
C01376=1219.078,93.968,-47.956,-178.597,5.636,148.572
C01377=1219.082,93.718,-47.938,-178.600,5.635,148.572
C01378=1219.087,93.469,-47.920,-178.603,5.634,148.573
C01379=1219.093,93.220,-47.901,-178.605,5.633,148.573
C01380=1219.097,92.971,-47.882,-178.608,5.632,148.574
C01381=1219.102,92.721,-47.864,-178.610,5.631,148.575
C01382=1219.106,92.472,-47.846,-178.613,5.631,148.575
C01383=1219.111,92.223,-47.828,-178.616,5.629,148.576
C01384=1219.117,91.974,-47.809,-178.618,5.629,148.576
C01385=1219.121,91.724,-47.791,-178.621,5.628,148.577
C01386=1219.126,91.475,-47.773,-178.623,5.627,148.578
C01387=1219.131,91.226,-47.755,-178.625,5.626,148.578
C01388=1219.136,90.977,-47.737,-178.629,5.625,148.579
C01389=1219.140,90.727,-47.718,-178.631,5.624,148.579
C01390=1219.146,90.477,-47.700,-178.633,5.623,148.580
C01391=1219.150,90.229,-47.681,-178.636,5.623,148.580
C01392=1219.155,89.980,-47.663,-178.638,5.622,148.581
C01393=1219.160,89.730,-47.645,-178.641,5.621,148.581
C01394=1219.164,89.481,-47.627,-178.644,5.620,148.582
C01395=1219.169,89.231,-47.609,-178.646,5.619,148.583
C01396=1219.174,88.982,-47.591,-178.649,5.618,148.583
C01397=1219.179,88.733,-47.573,-178.651,5.618,148.584
C01398=1219.184,88.484,-47.555,-178.654,5.617,148.584
C01399=1219.189,88.234,-47.536,-178.657,5.615,148.585
C01400=1219.194,87.984,-47.518,-178.659,5.615,148.586
C01401=1219.199,87.735,-47.500,-178.662,5.614,148.586
C01402=1219.204,87.486,-47.482,-178.664,5.614,148.587
C01403=1219.209,87.238,-47.463,-178.667,5.613,148.587
C01404=1219.213,86.988,-47.445,-178.669,5.612,148.588
C01405=1219.218,86.739,-47.427,-178.672,5.611,148.589
C01406=1219.223,86.489,-47.409,-178.674,5.610,148.589
C01407=1219.228,86.240,-47.391,-178.677,5.609,148.590
C01408=1219.233,85.990,-47.374,-178.680,5.609,148.590
C01409=1219.238,85.741,-47.356,-178.682,5.608,148.591
C01410=1219.243,85.492,-47.338,-178.684,5.607,148.591
C01411=1219.248,85.243,-47.320,-178.688,5.606,148.592
C01412=1219.252,84.993,-47.301,-178.690,5.605,148.592
C01413=1219.257,84.744,-47.283,-178.692,5.604,148.593
C01414=1219.262,84.495,-47.265,-178.695,5.604,148.594
C01415=1219.267,84.245,-47.247,-178.698,5.603,148.594
C01416=1219.271,83.996,-47.229,-178.700,5.602,148.595
C01417=1219.276,83.747,-47.211,-178.703,5.601,148.595
C01418=1219.281,83.498,-47.193,-178.706,5.600,148.596
C01419=1219.286,83.249,-47.175,-178.708,5.599,148.597
C01420=1219.291,83.000,-47.157,-178.710,5.599,148.597
C01421=1219.296,82.749,-47.140,-178.713,5.598,148.598
C01422=1219.301,82.500,-47.122,-178.715,5.597,148.598
C01423=1219.306,82.251,-47.104,-178.718,5.596,148.599
C01424=1219.310,82.002,-47.086,-178.721,5.595,148.600
C01425=1219.316,81.733,-47.067,-178.724,5.594,148.600
C01426=1219.321,81.464,-47.048,-178.726,5.594,148.601
C01427=1219.326,81.196,-47.028,-178.729,5.593,148.602
C01428=1219.332,80.929,-47.009,-178.732,5.592,148.602
C01429=1219.336,80.679,-46.991,-178.734,5.591,148.603
C01430=1219.341,80.429,-46.974,-178.737,5.590,148.603
C01431=1219.346,80.180,-46.956,-178.739,5.590,148.604
C01432=1219.351,79.931,-46.938,-178.742,5.589,148.604
C01433=1219.356,79.681,-46.920,-178.744,5.588,148.605
C01434=1219.360,79.432,-46.903,-178.747,5.587,148.606
C01435=1219.365,79.183,-46.885,-178.750,5.586,148.606
C01436=1219.370,78.934,-46.867,-178.752,5.585,148.607
C01437=1219.375,78.684,-46.849,-178.755,5.585,148.607
C01438=1219.380,78.435,-46.832,-178.757,5.584,148.608
C01439=1219.385,78.185,-46.814,-178.759,5.583,148.608
C01440=1219.390,77.936,-46.796,-178.762,5.583,148.609
C01441=1219.395,77.687,-46.779,-178.765,5.582,148.610
C01442=1219.400,77.438,-46.761,-178.768,5.581,148.610
C01443=1219.405,77.188,-46.743,-178.770,5.580,148.611
C01444=1219.410,76.939,-46.726,-178.773,5.579,148.612
C01445=1219.415,76.689,-46.708,-178.775,5.579,148.612
C01446=1219.419,76.441,-46.691,-178.778,5.578,148.613
C01447=1219.424,76.191,-46.673,-178.780,5.577,148.613
C01448=1219.429,75.942,-46.655,-178.783,5.576,148.614
C01449=1219.434,75.692,-46.637,-178.785,5.576,148.615
C01450=1219.439,75.443,-46.620,-178.788,5.575,148.615
C01451=1219.443,75.194,-46.603,-178.791,5.574,148.616
C01452=1219.449,74.944,-46.586,-178.793,5.573,148.616
C01453=1219.453,74.695,-46.568,-178.796,5.572,148.617
C01454=1219.459,74.445,-46.550,-178.798,5.571,148.617
C01455=1219.463,74.196,-46.533,-178.801,5.571,148.618
C01456=1219.468,73.947,-46.515,-178.803,5.570,148.619
C01457=1219.473,73.697,-46.498,-178.806,5.570,148.619
C01458=1219.478,73.448,-46.480,-178.808,5.569,148.620
C01459=1219.483,73.199,-46.463,-178.811,5.568,148.620
C01460=1219.488,72.950,-46.445,-178.813,5.568,148.621
C01461=1219.493,72.700,-46.428,-178.817,5.566,148.622
C01462=1219.497,72.451,-46.411,-178.819,5.565,148.622
C01463=1219.502,72.202,-46.394,-178.821,5.565,148.623
C01464=1219.507,71.952,-46.376,-178.824,5.564,148.624
C01465=1219.513,71.703,-46.358,-178.827,5.564,148.624
C01466=1219.517,71.454,-46.341,-178.829,5.563,148.625
C01467=1219.522,71.204,-46.324,-178.831,5.562,148.625
C01468=1219.527,70.955,-46.306,-178.834,5.561,148.626
C01469=1219.531,70.705,-46.289,-178.837,5.561,148.627
C01470=1219.537,70.455,-46.272,-178.839,5.560,148.627
C01471=1219.542,70.207,-46.254,-178.841,5.559,148.628
C01472=1219.547,69.958,-46.237,-178.845,5.558,148.628
C01473=1219.551,69.708,-46.219,-178.847,5.557,148.629
C01474=1219.556,69.459,-46.203,-178.850,5.557,148.630
C01475=1219.561,69.209,-46.186,-178.852,5.556,148.630
C01476=1219.566,68.960,-46.168,-178.855,5.555,148.631
C01477=1219.571,68.710,-46.151,-178.857,5.555,148.631
C01478=1219.575,68.461,-46.133,-178.860,5.554,148.632
C01479=1219.580,68.212,-46.116,-178.862,5.553,148.633
C01480=1219.586,67.963,-46.099,-178.865,5.553,148.633
C01481=1219.591,67.714,-46.081,-178.867,5.552,148.634
C01482=1219.595,67.464,-46.065,-178.870,5.552,148.635
C01483=1219.600,67.214,-46.047,-178.872,5.551,148.635
C01484=1219.605,66.965,-46.030,-178.875,5.550,148.636
C01485=1219.610,66.716,-46.013,-178.877,5.549,148.636
C01486=1219.615,66.467,-45.996,-178.880,5.549,148.637
C01487=1219.620,66.217,-45.979,-178.883,5.548,148.638
C01488=1219.625,65.968,-45.961,-178.885,5.547,148.638
C01489=1219.629,65.718,-45.945,-178.888,5.546,148.639
C01490=1219.635,65.469,-45.927,-178.891,5.545,148.639
C01491=1219.639,65.220,-45.910,-178.893,5.545,148.640
C01492=1219.645,64.971,-45.893,-178.895,5.544,148.640
C01493=1219.649,64.721,-45.876,-178.898,5.543,148.641
C01494=1219.654,64.471,-45.859,-178.901,5.543,148.642
C01495=1219.659,64.222,-45.842,-178.903,5.542,148.642
C01496=1219.664,63.973,-45.824,-178.906,5.542,148.643
C01497=1219.669,63.724,-45.808,-178.908,5.541,148.644
C01498=1219.674,63.474,-45.791,-178.911,5.540,148.644
C01499=1219.679,63.225,-45.774,-178.913,5.540,148.645
C01500=1219.684,62.975,-45.757,-178.916,5.539,148.646
C01501=1219.688,62.726,-45.740,-178.918,5.538,148.646
C01502=1219.694,62.477,-45.723,-178.921,5.538,148.647
C01503=1219.698,62.227,-45.706,-178.923,5.537,148.647
C01504=1219.703,61.978,-45.689,-178.926,5.536,148.648
C01505=1219.708,61.728,-45.672,-178.929,5.536,148.649
C01506=1219.713,61.479,-45.656,-178.931,5.535,148.649
C01507=1219.718,61.229,-45.638,-178.934,5.534,148.650
C01508=1219.723,60.980,-45.622,-178.937,5.533,148.650
C01509=1219.728,60.731,-45.604,-178.939,5.532,148.651
C01510=1219.733,60.482,-45.588,-178.942,5.532,148.652
C01511=1219.738,60.232,-45.570,-178.944,5.531,148.652
C01512=1219.742,59.983,-45.554,-178.947,5.530,148.653
C01513=1219.747,59.733,-45.537,-178.949,5.530,148.653
C01514=1219.753,59.484,-45.520,-178.952,5.529,148.654
C01515=1219.757,59.235,-45.503,-178.954,5.529,148.655
C01516=1219.762,58.985,-45.487,-178.957,5.528,148.655
C01517=1219.768,58.736,-45.470,-178.959,5.527,148.656
C01518=1219.772,58.487,-45.453,-178.962,5.527,148.657
C01519=1219.777,58.237,-45.436,-178.964,5.526,148.657
C01520=1219.782,57.987,-45.419,-178.967,5.525,148.658
C01521=1219.787,57.739,-45.403,-178.969,5.525,148.658
C01522=1219.792,57.489,-45.386,-178.972,5.524,148.659
C01523=1219.796,57.239,-45.369,-178.975,5.523,148.660
C01524=1219.802,56.991,-45.353,-178.977,5.523,148.660
C01525=1219.807,56.741,-45.335,-178.980,5.522,148.661
C01526=1219.811,56.491,-45.319,-178.982,5.521,148.661
C01527=1219.816,56.242,-45.302,-178.985,5.521,148.662
C01528=1219.822,55.993,-45.285,-178.987,5.520,148.663
C01529=1219.826,55.723,-45.268,-178.990,5.520,148.663
C01530=1219.832,55.456,-45.250,-178.992,5.519,148.664
C01531=1219.838,55.187,-45.232,-178.995,5.519,148.665
C01532=1219.842,54.919,-45.214,-178.998,5.517,148.665
C01533=1219.847,54.669,-45.197,-179.001,5.517,148.666
C01534=1219.853,54.420,-45.181,-179.004,5.516,148.667
C01535=1219.857,54.170,-45.164,-179.006,5.515,148.667
C01536=1219.863,53.921,-45.148,-179.009,5.515,148.668
C01537=1219.867,53.672,-45.131,-179.011,5.514,148.669
C01538=1219.872,53.422,-45.114,-179.014,5.513,148.669
C01539=1219.877,53.173,-45.098,-179.016,5.513,148.670
C01540=1219.882,52.923,-45.082,-179.019,5.512,148.671
C01541=1219.887,52.674,-45.065,-179.022,5.512,148.671
C01542=1219.892,52.425,-45.048,-179.024,5.511,148.672
C01543=1219.897,52.175,-45.031,-179.026,5.510,148.672
C01544=1219.901,51.926,-45.015,-179.029,5.510,148.673
C01545=1219.907,51.676,-44.999,-179.032,5.509,148.674
C01546=1219.911,51.427,-44.982,-179.034,5.509,148.674
C01547=1219.917,51.178,-44.966,-179.037,5.508,148.675
C01548=1219.922,50.928,-44.949,-179.039,5.507,148.675
C01549=1219.926,50.679,-44.932,-179.042,5.507,148.676
C01550=1219.931,50.429,-44.917,-179.044,5.506,148.677
C01551=1219.936,50.180,-44.900,-179.047,5.505,148.677
C01552=1219.941,49.931,-44.884,-179.049,5.506,148.678
C01553=1219.946,49.681,-44.867,-179.052,5.505,148.679
C01554=1219.952,49.432,-44.851,-179.054,5.504,148.679
C01555=1219.956,49.182,-44.834,-179.056,5.504,148.680
C01556=1219.961,48.933,-44.817,-179.059,5.503,148.681
C01557=1219.966,48.684,-44.802,-179.062,5.503,148.681
C01558=1219.970,48.434,-44.785,-179.064,5.502,148.682
C01559=1219.975,48.185,-44.769,-179.067,5.501,148.683
C01560=1219.981,47.935,-44.752,-179.069,5.500,148.683
C01561=1219.986,47.686,-44.736,-179.072,5.500,148.684
C01562=1219.991,47.437,-44.719,-179.074,5.499,148.684
C01563=1219.996,47.187,-44.704,-179.077,5.499,148.685
C01564=1220.000,46.938,-44.687,-179.080,5.498,148.686
C01565=1220.005,46.688,-44.671,-179.082,5.498,148.686
C01566=1220.010,46.439,-44.655,-179.085,5.497,148.687
C01567=1220.015,46.189,-44.638,-179.087,5.496,148.688
C01568=1220.020,45.940,-44.623,-179.090,5.496,148.688
C01569=1220.025,45.690,-44.606,-179.092,5.495,148.689
C01570=1220.030,45.441,-44.590,-179.095,5.495,148.690
C01571=1220.035,45.192,-44.574,-179.098,5.494,148.690
C01572=1220.040,44.943,-44.557,-179.100,5.493,148.691
C01573=1220.045,44.692,-44.541,-179.102,5.493,148.691
C01574=1220.050,44.444,-44.524,-179.105,5.492,148.692
C01575=1220.055,44.193,-44.509,-179.108,5.491,148.693
C01576=1220.060,43.945,-44.492,-179.110,5.491,148.693
C01577=1220.065,43.695,-44.476,-179.113,5.490,148.694
C01578=1220.070,43.446,-44.460,-179.116,5.490,148.695
C01579=1220.075,43.196,-44.444,-179.118,5.489,148.695
C01580=1220.080,42.947,-44.428,-179.120,5.489,148.696
C01581=1220.085,42.697,-44.412,-179.122,5.489,148.696
C01582=1220.090,42.448,-44.395,-179.125,5.488,148.697
C01583=1220.095,42.199,-44.380,-179.128,5.487,148.698
C01584=1220.100,41.949,-44.363,-179.130,5.487,148.698
C01585=1220.105,41.700,-44.348,-179.133,5.486,148.699
C01586=1220.110,41.450,-44.332,-179.136,5.486,148.700
C01587=1220.115,41.201,-44.315,-179.138,5.485,148.700
C01588=1220.119,40.951,-44.300,-179.140,5.484,148.701
C01589=1220.124,40.702,-44.284,-179.143,5.484,148.702
C01590=1220.129,40.452,-44.268,-179.146,5.483,148.702
C01591=1220.134,40.203,-44.251,-179.148,5.483,148.703
C01592=1220.139,39.954,-44.236,-179.151,5.482,148.704
C01593=1220.144,39.704,-44.220,-179.154,5.482,148.704
C01594=1220.149,39.455,-44.204,-179.156,5.481,148.705
C01595=1220.154,39.205,-44.188,-179.158,5.480,148.705
C01596=1220.159,38.956,-44.172,-179.161,5.480,148.706
C01597=1220.164,38.707,-44.156,-179.163,5.480,148.707
C01598=1220.169,38.457,-44.140,-179.166,5.479,148.707
C01599=1220.174,38.207,-44.124,-179.168,5.479,148.708
C01600=1220.179,37.958,-44.108,-179.171,5.478,148.709
C01601=1220.184,37.709,-44.093,-179.174,5.478,148.709
C01602=1220.189,37.459,-44.077,-179.176,5.477,148.710
C01603=1220.193,37.210,-44.060,-179.179,5.476,148.711
C01604=1220.199,36.960,-44.045,-179.181,5.476,148.711
C01605=1220.204,36.710,-44.029,-179.184,5.475,148.712
C01606=1220.209,36.461,-44.013,-179.186,5.475,148.713
C01607=1220.214,36.212,-43.997,-179.189,5.474,148.713
C01608=1220.218,35.962,-43.981,-179.192,5.473,148.714
C01609=1220.224,35.713,-43.966,-179.194,5.474,148.715
C01610=1220.229,35.464,-43.950,-179.196,5.473,148.715
C01611=1220.233,35.214,-43.934,-179.199,5.472,148.716
C01612=1220.239,34.965,-43.918,-179.201,5.472,148.716
C01613=1220.244,34.715,-43.902,-179.204,5.471,148.717
C01614=1220.248,34.465,-43.887,-179.207,5.471,148.718
C01615=1220.253,34.217,-43.871,-179.209,5.470,148.718
C01616=1220.259,33.967,-43.855,-179.212,5.470,148.719
C01617=1220.263,33.717,-43.839,-179.214,5.469,148.720
C01618=1220.269,33.468,-43.824,-179.217,5.468,148.721
C01619=1220.274,33.219,-43.809,-179.219,5.468,148.721
C01620=1220.278,32.969,-43.793,-179.221,5.468,148.722
C01621=1220.283,32.720,-43.776,-179.224,5.467,148.722
C01622=1220.289,32.470,-43.761,-179.227,5.467,148.723
C01623=1220.293,32.221,-43.745,-179.229,5.466,148.724
C01624=1220.298,31.971,-43.730,-179.232,5.466,148.724
C01625=1220.304,31.722,-43.714,-179.235,5.465,148.725
C01626=1220.308,31.472,-43.698,-179.237,5.465,148.726
C01627=1220.313,31.223,-43.683,-179.240,5.464,148.726
C01628=1220.318,30.973,-43.668,-179.242,5.463,148.727
C01629=1220.323,30.724,-43.651,-179.245,5.463,148.727
C01630=1220.328,30.475,-43.636,-179.247,5.463,148.728
C01631=1220.333,30.225,-43.621,-179.249,5.462,148.729
C01632=1220.338,29.976,-43.605,-179.252,5.462,148.730
C01633=1220.343,29.707,-43.588,-179.255,5.461,148.730
C01634=1220.348,29.438,-43.572,-179.257,5.461,148.731
C01635=1220.354,29.169,-43.555,-179.260,5.460,148.732
C01636=1220.360,28.901,-43.538,-179.263,5.460,148.732
C01637=1220.364,28.652,-43.523,-179.265,5.459,148.733
C01638=1220.370,28.402,-43.507,-179.268,5.459,148.734
C01639=1220.374,28.152,-43.491,-179.270,5.458,148.734
C01640=1220.379,27.903,-43.476,-179.273,5.457,148.735
C01641=1220.384,27.654,-43.461,-179.276,5.457,148.736
C01642=1220.390,27.404,-43.445,-179.278,5.456,148.736
C01643=1220.394,27.155,-43.430,-179.281,5.456,148.737
C01644=1220.399,26.905,-43.414,-179.283,5.456,148.738
C01645=1220.405,26.656,-43.399,-179.286,5.456,148.738
C01646=1220.409,26.407,-43.384,-179.288,5.455,148.739
C01647=1220.414,26.156,-43.368,-179.291,5.454,148.739
C01648=1220.419,25.907,-43.353,-179.293,5.454,148.740
C01649=1220.424,25.657,-43.338,-179.296,5.453,148.741
C01650=1220.430,25.408,-43.322,-179.299,5.453,148.742
C01651=1220.434,25.159,-43.307,-179.301,5.452,148.742
C01652=1220.439,24.909,-43.291,-179.303,5.452,148.743
C01653=1220.444,24.660,-43.276,-179.306,5.452,148.744
C01654=1220.449,24.410,-43.261,-179.309,5.451,148.744
C01655=1220.455,24.161,-43.245,-179.311,5.451,148.745
C01656=1220.459,23.912,-43.230,-179.314,5.450,148.746
C01657=1220.464,23.661,-43.215,-179.316,5.449,148.746
C01658=1220.469,23.412,-43.200,-179.319,5.449,148.747
C01659=1220.474,23.163,-43.184,-179.321,5.449,148.747
C01660=1220.479,22.914,-43.169,-179.323,5.448,148.748
C01661=1220.484,22.664,-43.154,-179.326,5.448,148.749
C01662=1220.489,22.415,-43.139,-179.329,5.447,148.749
C01663=1220.494,22.164,-43.123,-179.331,5.447,148.750
C01664=1220.499,21.915,-43.108,-179.334,5.446,148.751
C01665=1220.504,21.666,-43.093,-179.337,5.446,148.751
C01666=1220.509,21.417,-43.078,-179.339,5.446,148.752
C01667=1220.514,21.167,-43.062,-179.341,5.445,148.753
C01668=1220.519,20.918,-43.048,-179.344,5.445,148.754
C01669=1220.525,20.668,-43.032,-179.346,5.444,148.754
C01670=1220.529,20.418,-43.017,-179.349,5.444,148.755
C01671=1220.534,20.169,-43.001,-179.351,5.443,148.755
C01672=1220.539,19.919,-42.987,-179.354,5.442,148.756
C01673=1220.544,19.670,-42.972,-179.356,5.443,148.757
C01674=1220.549,19.421,-42.957,-179.359,5.442,148.757
C01675=1220.555,19.171,-42.942,-179.361,5.442,148.758
C01676=1220.559,18.922,-42.927,-179.364,5.441,148.759
C01677=1220.565,18.672,-42.911,-179.367,5.441,148.759
C01678=1220.569,18.423,-42.896,-179.369,5.440,148.760
C01679=1220.574,18.173,-42.882,-179.371,5.440,148.761
C01680=1220.579,17.923,-42.866,-179.374,5.440,148.762
C01681=1220.584,17.674,-42.851,-179.377,5.439,148.762
C01682=1220.589,17.424,-42.836,-179.379,5.438,148.763
C01683=1220.594,17.175,-42.821,-179.381,5.438,148.763
C01684=1220.600,16.925,-42.806,-179.384,5.437,148.764
C01685=1220.604,16.676,-42.791,-179.386,5.438,148.765
C01686=1220.609,16.427,-42.776,-179.389,5.437,148.765
C01687=1220.615,16.177,-42.761,-179.392,5.437,148.766
C01688=1220.619,15.928,-42.746,-179.394,5.436,148.767
C01689=1220.624,15.679,-42.731,-179.397,5.435,148.767
C01690=1220.629,15.428,-42.716,-179.399,5.435,148.768
C01691=1220.634,15.179,-42.701,-179.402,5.435,148.769
C01692=1220.640,14.929,-42.686,-179.404,5.435,148.769
C01693=1220.644,14.680,-42.671,-179.407,5.434,148.770
C01694=1220.649,14.430,-42.657,-179.409,5.434,148.771
C01695=1220.655,14.181,-42.641,-179.412,5.433,148.771
C01696=1220.659,13.932,-42.626,-179.414,5.432,148.772
C01697=1220.664,13.682,-42.612,-179.416,5.433,148.773
C01698=1220.669,13.433,-42.597,-179.419,5.432,148.773
C01699=1220.674,13.183,-42.582,-179.422,5.431,148.774
C01700=1220.679,12.934,-42.567,-179.424,5.431,148.775
C01701=1220.685,12.684,-42.552,-179.427,5.430,148.775
C01702=1220.689,12.435,-42.537,-179.429,5.431,148.776
C01703=1220.694,12.185,-42.523,-179.432,5.430,148.777
C01704=1220.699,11.936,-42.508,-179.434,5.430,148.777
C01705=1220.705,11.686,-42.493,-179.437,5.429,148.778
C01706=1220.709,11.437,-42.478,-179.440,5.429,148.779
C01707=1220.714,11.187,-42.464,-179.442,5.429,148.780
C01708=1220.720,10.937,-42.449,-179.444,5.428,148.780
C01709=1220.725,10.688,-42.434,-179.447,5.428,148.781
C01710=1220.730,10.438,-42.420,-179.450,5.427,148.782
C01711=1220.734,10.189,-42.405,-179.452,5.426,148.782
C01712=1220.740,9.939,-42.390,-179.454,5.426,148.783
C01713=1220.745,9.690,-42.375,-179.457,5.426,148.783
C01714=1220.750,9.440,-42.361,-179.459,5.426,148.784
C01715=1220.755,9.191,-42.346,-179.462,5.425,148.785
C01716=1220.759,8.942,-42.331,-179.464,5.425,148.785
C01717=1220.765,8.691,-42.317,-179.467,5.424,148.786
C01718=1220.770,8.442,-42.302,-179.469,5.424,148.787
C01719=1220.774,8.193,-42.287,-179.472,5.424,148.788
C01720=1220.779,7.943,-42.273,-179.474,5.423,148.788
C01721=1220.784,7.694,-42.258,-179.477,5.423,148.789
C01722=1220.790,7.444,-42.243,-179.480,5.422,148.790
C01723=1220.795,7.195,-42.229,-179.482,5.423,148.790
C01724=1220.800,6.945,-42.215,-179.485,5.422,148.791
C01725=1220.805,6.696,-42.200,-179.487,5.422,148.792
C01726=1220.810,6.446,-42.186,-179.490,5.421,148.792
C01727=1220.816,6.196,-42.171,-179.492,5.421,148.793
C01728=1220.820,5.947,-42.156,-179.495,5.421,148.794
C01729=1220.825,5.698,-42.142,-179.497,5.420,148.794
C01730=1220.830,5.448,-42.127,-179.499,5.419,148.795
C01731=1220.835,5.199,-42.112,-179.502,5.419,148.796
C01732=1220.840,4.949,-42.098,-179.504,5.419,148.796
C01733=1220.845,4.699,-42.084,-179.507,5.419,148.797
C01734=1220.850,4.449,-42.069,-179.509,5.418,148.798
C01735=1220.855,4.200,-42.054,-179.512,5.418,148.798
C01736=1220.861,3.951,-42.040,-179.515,5.417,148.799
C01737=1220.866,3.682,-42.025,-179.517,5.417,148.800
C01738=1220.871,3.413,-42.009,-179.519,5.417,148.800
C01739=1220.876,3.144,-41.994,-179.523,5.417,148.801
C01740=1220.881,2.875,-41.978,-179.525,5.416,148.802
C01741=1220.887,2.625,-41.963,-179.528,5.416,148.803
C01742=1220.892,2.376,-41.949,-179.531,5.415,148.803
C01743=1220.897,2.126,-41.934,-179.533,5.415,148.804
C01744=1220.903,1.877,-41.921,-179.535,5.415,148.805
C01745=1220.908,1.627,-41.906,-179.538,5.414,148.805
C01746=1220.912,1.378,-41.891,-179.541,5.414,148.806
C01747=1220.917,1.128,-41.877,-179.543,5.413,148.807
C01748=1220.922,0.879,-41.863,-179.545,5.413,148.807
C01749=1220.927,0.629,-41.848,-179.547,5.413,148.808
C01750=1220.932,0.379,-41.834,-179.550,5.412,148.809
C01751=1220.938,0.130,-41.820,-179.553,5.412,148.809
C01752=1220.943,-0.119,-41.806,-179.555,5.412,148.810
C01753=1220.947,-0.369,-41.792,-179.557,5.412,148.811
C01754=1220.952,-0.619,-41.777,-179.560,5.411,148.811
C01755=1220.957,-0.869,-41.763,-179.563,5.410,148.812
C01756=1220.963,-1.117,-41.748,-179.565,5.410,148.813
C01757=1220.968,-1.367,-41.734,-179.568,5.410,148.813
C01758=1220.973,-1.616,-41.720,-179.570,5.410,148.814
C01759=1220.977,-1.866,-41.706,-179.573,5.409,148.815
C01760=1220.982,-2.116,-41.691,-179.575,5.409,148.815
C01761=1220.987,-2.366,-41.677,-179.578,5.409,148.816
C01762=1220.993,-2.615,-41.663,-179.580,5.408,148.817
C01763=1220.998,-2.864,-41.649,-179.583,5.408,148.818
C01764=1221.003,-3.114,-41.635,-179.586,5.407,148.818
C01765=1221.008,-3.364,-41.620,-179.588,5.408,148.819
C01766=1221.013,-3.613,-41.606,-179.590,5.407,148.820
C01767=1221.018,-3.862,-41.592,-179.593,5.407,148.820
C01768=1221.023,-4.112,-41.578,-179.596,5.406,148.821
C01769=1221.028,-4.362,-41.564,-179.598,5.407,148.822
C01770=1221.033,-4.612,-41.549,-179.600,5.406,148.822
C01771=1221.039,-4.861,-41.535,-179.603,5.406,148.823
C01772=1221.043,-5.110,-41.522,-179.605,5.405,148.824
C01773=1221.048,-5.360,-41.507,-179.607,5.405,148.824
C01774=1221.053,-5.610,-41.494,-179.610,5.404,148.825
C01775=1221.059,-5.859,-41.480,-179.613,5.404,148.826
C01776=1221.064,-6.109,-41.466,-179.615,5.403,148.826
C01777=1221.069,-6.358,-41.451,-179.617,5.404,148.827
C01778=1221.074,-6.608,-41.437,-179.620,5.403,148.828
C01779=1221.079,-6.857,-41.423,-179.623,5.403,148.828
C01780=1221.083,-7.106,-41.410,-179.625,5.402,148.829
C01781=1221.088,-7.356,-41.395,-179.627,5.402,148.830
C01782=1221.093,-7.606,-41.381,-179.630,5.402,148.830
C01783=1221.099,-7.856,-41.368,-179.633,5.401,148.831
C01784=1221.104,-8.105,-41.354,-179.635,5.401,148.832
C01785=1221.109,-8.355,-41.339,-179.637,5.401,148.833
C01786=1221.115,-8.604,-41.325,-179.640,5.401,148.833
C01787=1221.119,-8.853,-41.312,-179.643,5.400,148.834
C01788=1221.124,-9.103,-41.297,-179.645,5.401,148.835
C01789=1221.129,-9.353,-41.284,-179.647,5.400,148.835
C01790=1221.135,-9.602,-41.270,-179.650,5.399,148.836
C01791=1221.140,-9.852,-41.256,-179.653,5.399,148.837
C01792=1221.144,-10.102,-41.242,-179.655,5.399,148.837
C01793=1221.149,-10.351,-41.228,-179.657,5.399,148.838
C01794=1221.155,-10.601,-41.214,-179.660,5.398,148.839
C01795=1221.160,-10.851,-41.200,-179.663,5.398,148.839
C01796=1221.165,-11.100,-41.186,-179.665,5.398,148.840
C01797=1221.169,-11.349,-41.173,-179.667,5.398,148.841
C01798=1221.175,-11.599,-41.159,-179.670,5.397,148.842
C01799=1221.180,-11.848,-41.145,-179.672,5.397,148.842
C01800=1221.185,-12.098,-41.131,-179.675,5.397,148.843
C01801=1221.189,-12.347,-41.117,-179.678,5.396,148.844
C01802=1221.195,-12.597,-41.104,-179.680,5.396,148.844
C01803=1221.200,-12.847,-41.090,-179.682,5.396,148.845
C01804=1221.205,-13.096,-41.075,-179.684,5.395,148.845
C01805=1221.210,-13.346,-41.063,-179.687,5.395,148.846
C01806=1221.215,-13.596,-41.049,-179.689,5.395,148.847
C01807=1221.220,-13.845,-41.034,-179.692,5.395,148.848
C01808=1221.226,-14.095,-41.021,-179.694,5.394,148.848
C01809=1221.230,-14.344,-41.007,-179.697,5.394,148.849
C01810=1221.236,-14.593,-40.993,-179.699,5.394,148.850
C01811=1221.241,-14.844,-40.980,-179.702,5.393,148.850
C01812=1221.245,-15.093,-40.966,-179.705,5.393,148.851
C01813=1221.251,-15.342,-40.952,-179.707,5.393,148.852
C01814=1221.256,-15.592,-40.939,-179.709,5.393,148.852
C01815=1221.260,-15.842,-40.925,-179.712,5.392,148.853
C01816=1221.266,-16.091,-40.911,-179.715,5.392,148.854
C01817=1221.271,-16.341,-40.898,-179.717,5.392,148.854
C01818=1221.276,-16.590,-40.884,-179.719,5.391,148.855
